LIN {X 0,Y 425.288,Z 130.32,A -85,B 0,C 180,E1 -9761.958,E2 -9761.958} C_VEL
LIN {X 0,Y 425.283,Z 130.319,A -85,B 0,C 180,E1 -9765.283,E2 -9765.283} C_VEL
LIN {X 0,Y 425.272,Z 130.322,A -85,B 0,C 180,E1 -9768.622,E2 -9768.622} C_VEL
LIN {X 0,Y 425.304,Z 130.316,A -85,B 0,C 180,E1 -9771.102,E2 -9771.102} C_VEL
LIN {X 0,Y 425.298,Z 130.317,A -85,B 0,C 180,E1 -9774.664,E2 -9774.664} C_VEL
LIN {X 0,Y 425.263,Z 130.324,A -85,B 0,C 180,E1 -9778.073,E2 -9778.073} C_VEL
LIN {X 0,Y 425.33,Z 130.317,A -85,B 0,C 180,E1 -9781.368,E2 -9781.368} C_VEL
LIN {X 0,Y 425.295,Z 130.314,A -85,B 0,C 180,E1 -9784.555,E2 -9784.555} C_VEL
LIN {X 0,Y 425.395,Z 130.501,A -85,B 0,C 180,E1 -9786.124,E2 -9786.124} C_VEL
LIN {X 0,Y 426.718,Z 138.86,A -85,B 0,C 180,E1 -9788.249,E2 -9788.249} C_VEL
LIN {X 0,Y 426.399,Z 147.655,A -85,B 0,C 180,E1 -9790.343,E2 -9790.343} C_VEL
LIN {X 0,Y 425.564,Z 164.044,A -85,B 0,C 180,E1 -9794.188,E2 -9794.188} C_VEL
LIN {X 0,Y 425.386,Z 168.668,A -85,B 0,C 180,E1 -9795.224,E2 -9795.224} C_VEL
LIN {X 0,Y 425.881,Z 172.494,A -85,B 0,C 180,E1 -9795.359,E2 -9795.359} C_VEL
LIN {X 0,Y 428.081,Z 189.094,A -85,B 0,C 180,E1 -9795.717,E2 -9795.717} C_VEL
LIN {X 0,Y 427.768,Z 244.774,A -85,B 0,C 180,E1 -9796.671,E2 -9796.671} C_VEL
LIN {X 0,Y 427.448,Z 254.051,A -85,B 0,C 180,E1 -9796.934,E2 -9796.934} C_VEL
LIN {X 0,Y 427.1,Z 263.713,A -85,B 0,C 180,E1 -9797.346,E2 -9797.346} C_VEL
LIN {X 0,Y 426.691,Z 272.874,A -85,B 0,C 180,E1 -9797.878,E2 -9797.878} C_VEL
LIN {X 0,Y 426.182,Z 283.679,A -85,B 0,C 180,E1 -9798.707,E2 -9798.707} C_VEL
LIN {X 0,Y 425.644,Z 292.988,A -85,B 0,C 180,E1 -9799.656,E2 -9799.656} C_VEL
LIN {X 0,Y 425.305,Z 299.661,A -85,B 0,C 180,E1 -9800.489,E2 -9800.489} C_VEL
LIN {X 0,Y 424.937,Z 305.994,A -85,B 0,C 180,E1 -9801.44,E2 -9801.44} C_VEL
LIN {X 0,Y 424.669,Z 311.256,A -85,B 0,C 180,E1 -9802.392,E2 -9802.392} C_VEL
LIN {X 0,Y 424.421,Z 316.205,A -85,B 0,C 180,E1 -9803.484,E2 -9803.484} C_VEL
LIN {X 0,Y 424.283,Z 320.82,A -85,B 0,C 180,E1 -9804.773,E2 -9804.773} C_VEL
LIN {X 0,Y 424.129,Z 324.618,A -85,B 0,C 180,E1 -9806.2,E2 -9806.2} C_VEL
LIN {X 0,Y 424.106,Z 326.365,A -85,B 0,C 180,E1 -9807.151,E2 -9807.151} C_VEL
LIN {X 0,Y 424.122,Z 327.617,A -85,B 0,C 180,E1 -9808.101,E2 -9808.101} C_VEL
LIN {X 0,Y 424.067,Z 328.395,A -85,B 0,C 180,E1 -9809.051,E2 -9809.051} C_VEL
LIN {X 0,Y 424.06,Z 328.689,A -85,B 0,C 180,E1 -9810,E2 -9810} C_VEL
LIN {X 0,Y 424.067,Z 328.392,A -85,B 0,C 180,E1 -9810.95,E2 -9810.95} C_VEL
LIN {X 0,Y 424.122,Z 327.61,A -85,B 0,C 180,E1 -9811.899,E2 -9811.899} C_VEL
LIN {X 0,Y 424.106,Z 326.354,A -85,B 0,C 180,E1 -9812.85,E2 -9812.85} C_VEL
LIN {X 0,Y 424.165,Z 323.448,A -85,B 0,C 180,E1 -9814.276,E2 -9814.276} C_VEL
LIN {X 0,Y 424.283,Z 320.8,A -85,B 0,C 180,E1 -9815.227,E2 -9815.227} C_VEL
LIN {X 0,Y 424.459,Z 315.617,A -85,B 0,C 180,E1 -9816.656,E2 -9816.656} C_VEL
LIN {X 0,Y 424.748,Z 308.788,A -85,B 0,C 180,E1 -9818.085,E2 -9818.085} C_VEL
LIN {X 0,Y 425.194,Z 301.324,A -85,B 0,C 180,E1 -9819.274,E2 -9819.274} C_VEL
LIN {X 0,Y 425.588,Z 293.962,A -85,B 0,C 180,E1 -9820.226,E2 -9820.226} C_VEL
LIN {X 0,Y 426.052,Z 286.079,A -85,B 0,C 180,E1 -9821.056,E2 -9821.056} C_VEL
LIN {X 0,Y 426.49,Z 277.748,A -85,B 0,C 180,E1 -9821.767,E2 -9821.767} C_VEL
LIN {X 0,Y 426.99,Z 267.109,A -85,B 0,C 180,E1 -9822.476,E2 -9822.476} C_VEL
LIN {X 0,Y 427.37,Z 255.53,A -85,B 0,C 180,E1 -9823.008,E2 -9823.008} C_VEL
LIN {X 0,Y 427.68,Z 245.835,A -85,B 0,C 180,E1 -9823.301,E2 -9823.301} C_VEL
LIN {X 0,Y 428.097,Z 188.695,A -85,B 0,C 180,E1 -9824.283,E2 -9824.283} C_VEL
LIN {X 0,Y 425.376,Z 168.966,A -85,B 0,C 180,E1 -9824.74,E2 -9824.74} C_VEL
LIN {X 0,Y 425.469,Z 166.107,A -85,B 0,C 180,E1 -9825.325,E2 -9825.325} C_VEL
LIN {X 0,Y 426.143,Z 151.434,A -85,B 0,C 180,E1 -9828.76,E2 -9828.76} C_VEL
LIN {X 0,Y 426.783,Z 139.882,A -85,B 0,C 180,E1 -9831.494,E2 -9831.494} C_VEL
LIN {X 0,Y 426.048,Z 134.247,A -85,B 0,C 180,E1 -9832.894,E2 -9832.894} C_VEL
LIN {X 0,Y 425.366,Z 130.353,A -85,B 0,C 180,E1 -9833.943,E2 -9833.943} C_VEL
LIN {X 0,Y 425.349,Z 130.31,A -85,B 0,C 180,E1 -9837.558,E2 -9837.558} C_VEL
LIN {X 0,Y 425.288,Z 130.32,A -85,B 0,C 180,E1 -9840.816,E2 -9840.816} C_VEL
LIN {X 0,Y 425.312,Z 130.321,A -85,B 0,C 180,E1 -9844.288,E2 -9844.288} C_VEL
LIN {X 0,Y 425.279,Z 130.322,A -85,B 0,C 180,E1 -9847.694,E2 -9847.694} C_VEL
LIN {X 0,Y 425.28,Z 130.32,A -85,B 0,C 180,E1 -9850.52,E2 -9850.52} C_VEL
LIN {X 0,Y 425.257,Z 130.324,A -85,B 0,C 180,E1 -9853.351,E2 -9853.351} C_VEL
LIN {X 0,Y 425.257,Z 130.322,A -85,B 0,C 180,E1 -9856.649,E2 -9856.649} C_VEL
LIN {X 0,Y 425.286,Z 130.322,A -85,B 0,C 180,E1 -9859.873,E2 -9859.873} C_VEL
LIN {X 0,Y 425.278,Z 130.319,A -85,B 0,C 180,E1 -9862.489,E2 -9862.489} C_VEL
LIN {X 0,Y 425.309,Z 130.317,A -85,B 0,C 180,E1 -9865.818,E2 -9865.818} C_VEL
LIN {X 0,Y 425.291,Z 130.325,A -85,B 0,C 180,E1 -9869.239,E2 -9869.239} C_VEL
LIN {X 0,Y 425.35,Z 130.311,A -85,B 0,C 180,E1 -9872.442,E2 -9872.442} C_VEL
LIN {X 0,Y 425.352,Z 130.311,A -85,B 0,C 180,E1 -9875.602,E2 -9875.602} C_VEL
LIN {X 0,Y 425.294,Z 130.322,A -85,B 0,C 180,E1 -9878.682,E2 -9878.682} C_VEL
LIN {X 0,Y 425.334,Z 130.312,A -85,B 0,C 180,E1 -9881.703,E2 -9881.703} C_VEL
LIN {X 0,Y 425.35,Z 130.317,A -85,B 0,C 180,E1 -9884.671,E2 -9884.671} C_VEL
LIN {X 0,Y 425.413,Z 130.302,A -85,B 0,C 180,E1 -9887.598,E2 -9887.598} C_VEL
LIN {X 0,Y 425.444,Z 130.298,A -85,B 0,C 180,E1 -9891.45,E2 -9891.45} C_VEL
LIN {X 0,Y 425.552,Z 130.292,A -85,B 0,C 180,E1 -9894.313,E2 -9894.313} C_VEL
LIN {X 0,Y 425.575,Z 130.289,A -85,B 0,C 180,E1 -9898.107,E2 -9898.107} C_VEL
LIN {X 0,Y 425.703,Z 130.273,A -85,B 0,C 180,E1 -9900,E2 -9900} C_VEL
LIN {X 0,Y 425.547,Z 130.286,A -85,B 0,C 180,E1 -9902.84,E2 -9902.84} C_VEL
LIN {X 0,Y 425.533,Z 130.288,A -85,B 0,C 180,E1 -9906.639,E2 -9906.639} C_VEL
LIN {X 0,Y 425.405,Z 130.308,A -85,B 0,C 180,E1 -9909.509,E2 -9909.509} C_VEL
LIN {X 0,Y 425.406,Z 130.304,A -85,B 0,C 180,E1 -9912.91,E2 -9912.91} C_VEL
LIN {X 0,Y 425.363,Z 130.309,A -85,B 0,C 180,E1 -9916.605,E2 -9916.605} C_VEL
LIN {X 0,Y 425.33,Z 130.316,A -85,B 0,C 180,E1 -9919.636,E2 -9919.636} C_VEL
LIN {X 0,Y 425.308,Z 130.32,A -85,B 0,C 180,E1 -9923.365,E2 -9923.365} C_VEL
LIN {X 0,Y 425.349,Z 130.315,A -85,B 0,C 180,E1 -9926.844,E2 -9926.844} C_VEL
LIN {X 0,Y 425.293,Z 130.318,A -85,B 0,C 180,E1 -9929.72,E2 -9929.72} C_VEL
LIN {X 0,Y 425.284,Z 130.323,A -85,B 0,C 180,E1 -9933.048,E2 -9933.048} C_VEL
LIN {X 0,Y 425.285,Z 130.319,A -85,B 0,C 180,E1 -9935.929,E2 -9935.929} C_VEL
LIN {X 0,Y 425.283,Z 130.321,A -85,B 0,C 180,E1 -9939.041,E2 -9939.041} C_VEL
LIN {X 0,Y 425.291,Z 130.319,A -85,B 0,C 180,E1 -9941.958,E2 -9941.958} C_VEL
LIN {X 0,Y 425.286,Z 130.318,A -85,B 0,C 180,E1 -9945.283,E2 -9945.283} C_VEL
LIN {X 0,Y 425.277,Z 130.322,A -85,B 0,C 180,E1 -9948.622,E2 -9948.622} C_VEL
LIN {X 0,Y 425.317,Z 130.314,A -85,B 0,C 180,E1 -9951.103,E2 -9951.103} C_VEL
LIN {X 0,Y 425.302,Z 130.317,A -85,B 0,C 180,E1 -9954.664,E2 -9954.664} C_VEL
LIN {X 0,Y 425.267,Z 130.325,A -85,B 0,C 180,E1 -9958.073,E2 -9958.073} C_VEL
LIN {X 0,Y 425.333,Z 130.315,A -85,B 0,C 180,E1 -9961.368,E2 -9961.368} C_VEL
LIN {X 0,Y 425.355,Z 130.315,A -85,B 0,C 180,E1 -9963.505,E2 -9963.505} C_VEL
LIN {X 0,Y 425.287,Z 130.321,A -85,B 0,C 180,E1 -9966.634,E2 -9966.634} C_VEL
LIN {X 0,Y 425.375,Z 130.436,A -85,B 0,C 180,E1 -9969.13,E2 -9969.13} C_VEL
LIN {X 0,Y 426.152,Z 136.277,A -85,B 0,C 180,E1 -9970.741,E2 -9970.741} C_VEL
LIN {X 0,Y 425.734,Z 147.759,A -85,B 0,C 180,E1 -9973.702,E2 -9973.702} C_VEL
LIN {X 0,Y 425.508,Z 154.307,A -85,B 0,C 180,E1 -9975.298,E2 -9975.298} C_VEL
LIN {X 0,Y 426.018,Z 157.356,A -85,B 0,C 180,E1 -9975.412,E2 -9975.412} C_VEL
LIN {X 0,Y 428.175,Z 170.829,A -85,B 0,C 180,E1 -9975.717,E2 -9975.717} C_VEL
LIN {X 0,Y 427.787,Z 230.137,A -85,B 0,C 180,E1 -9976.733,E2 -9976.733} C_VEL
LIN {X 0,Y 427.576,Z 239.219,A -85,B 0,C 180,E1 -9976.998,E2 -9976.998} C_VEL
LIN {X 0,Y 427.327,Z 248.804,A -85,B 0,C 180,E1 -9977.413,E2 -9977.413} C_VEL
LIN {X 0,Y 426.923,Z 258.842,A -85,B 0,C 180,E1 -9978.004,E2 -9978.004} C_VEL
LIN {X 0,Y 426.381,Z 269.256,A -85,B 0,C 180,E1 -9978.833,E2 -9978.833} C_VEL
LIN {X 0,Y 425.985,Z 277.399,A -85,B 0,C 180,E1 -9979.664,E2 -9979.664} C_VEL
LIN {X 0,Y 425.58,Z 284.118,A -85,B 0,C 180,E1 -9980.494,E2 -9980.494} C_VEL
LIN {X 0,Y 425.466,Z 285.604,A -85,B 0,C 180,E1 -9980.702,E2 -9980.702} C_VEL
LIN {X 0,Y 424.548,Z 289.624,A -85,B 0,C 180,E1 -9981.28,E2 -9981.28} C_VEL
LIN {X 0,Y 420.037,Z 297.702,A -85,B 0,C 180,E1 -9982.687,E2 -9982.687} C_VEL
LIN {X 0,Y 417.925,Z 301.654,A -85,B 0,C 180,E1 -9983.579,E2 -9983.579} C_VEL
LIN {X 0,Y 417.506,Z 303.441,A -85,B 0,C 180,E1 -9984.055,E2 -9984.055} C_VEL
LIN {X 0,Y 417.267,Z 306.984,A -85,B 0,C 180,E1 -9985.169,E2 -9985.169} C_VEL
LIN {X 0,Y 417.172,Z 309.308,A -85,B 0,C 180,E1 -9986.136,E2 -9986.136} C_VEL
LIN {X 0,Y 417.127,Z 311.078,A -85,B 0,C 180,E1 -9987.102,E2 -9987.102} C_VEL
LIN {X 0,Y 417.064,Z 312.355,A -85,B 0,C 180,E1 -9988.068,E2 -9988.068} C_VEL
LIN {X 0,Y 416.993,Z 313.163,A -85,B 0,C 180,E1 -9989.034,E2 -9989.034} C_VEL
LIN {X 0,Y 416.983,Z 313.47,A -85,B 0,C 180,E1 -9990,E2 -9990} C_VEL
LIN {X 0,Y 416.993,Z 313.195,A -85,B 0,C 180,E1 -9990.965,E2 -9990.965} C_VEL
LIN {X 0,Y 417.064,Z 312.452,A -85,B 0,C 180,E1 -9991.931,E2 -9991.931} C_VEL
LIN {X 0,Y 417.125,Z 311.241,A -85,B 0,C 180,E1 -9992.897,E2 -9992.897} C_VEL
LIN {X 0,Y 417.2,Z 308.392,A -85,B 0,C 180,E1 -9994.347,E2 -9994.347} C_VEL
LIN {X 0,Y 417.362,Z 305.799,A -85,B 0,C 180,E1 -9995.314,E2 -9995.314} C_VEL
LIN {X 0,Y 417.669,Z 300.692,A -85,B 0,C 180,E1 -9996.764,E2 -9996.764} C_VEL
LIN {X 0,Y 417.888,Z 295.199,A -85,B 0,C 180,E1 -9997.975,E2 -9997.975} C_VEL
LIN {X 0,Y 418.33,Z 288.3,A -85,B 0,C 180,E1 -9999.183,E2 -9999.183} C_VEL
LIN {X 0,Y 418.819,Z 280.376,A -85,B 0,C 180,E1 -10000.27,E2 -10000.27} C_VEL
LIN {X 0,Y 419.251,Z 272.82,A -85,B 0,C 180,E1 -10001.115,E2 -10001.115} C_VEL
LIN {X 0,Y 419.666,Z 264.901,A -85,B 0,C 180,E1 -10001.838,E2 -10001.838} C_VEL
LIN {X 0,Y 420.075,Z 256.724,A -85,B 0,C 180,E1 -10002.439,E2 -10002.439} C_VEL
LIN {X 0,Y 420.443,Z 248.443,A -85,B 0,C 180,E1 -10002.919,E2 -10002.919} C_VEL
LIN {X 0,Y 420.771,Z 239.505,A -85,B 0,C 180,E1 -10003.308,E2 -10003.308} C_VEL
LIN {X 0,Y 420.957,Z 230.241,A -85,B 0,C 180,E1 -10003.585,E2 -10003.585} C_VEL
LIN {X 0,Y 421.276,Z 170.679,A -85,B 0,C 180,E1 -10004.626,E2 -10004.626} C_VEL
LIN {X 0,Y 418.531,Z 154.749,A -85,B 0,C 180,E1 -10005.024,E2 -10005.024} C_VEL
LIN {X 0,Y 418.508,Z 153.569,A -85,B 0,C 180,E1 -10005.211,E2 -10005.211} C_VEL
LIN {X 0,Y 419.078,Z 140.565,A -85,B 0,C 180,E1 -10008.58,E2 -10008.58} C_VEL
LIN {X 0,Y 418.969,Z 135.057,A -85,B 0,C 180,E1 -10010.053,E2 -10010.053} C_VEL
LIN {X 0,Y 418.322,Z 131.28,A -85,B 0,C 180,E1 -10011.174,E2 -10011.174} C_VEL
LIN {X 0,Y 418.285,Z 131.193,A -85,B 0,C 180,E1 -10014.864,E2 -10014.864} C_VEL
LIN {X 0,Y 418.292,Z 131.193,A -85,B 0,C 180,E1 -10018.063,E2 -10018.063} C_VEL
LIN {X 0,Y 418.211,Z 131.2,A -85,B 0,C 180,E1 -10021.396,E2 -10021.396} C_VEL
LIN {X 0,Y 418.266,Z 131.195,A -85,B 0,C 180,E1 -10024.58,E2 -10024.58} C_VEL
LIN {X 0,Y 418.234,Z 131.202,A -85,B 0,C 180,E1 -10027.834,E2 -10027.834} C_VEL
LIN {X 0,Y 418.223,Z 131.198,A -85,B 0,C 180,E1 -10030.948,E2 -10030.948} C_VEL
LIN {X 0,Y 418.21,Z 131.207,A -85,B 0,C 180,E1 -10033.729,E2 -10033.729} C_VEL
LIN {X 0,Y 418.207,Z 131.2,A -85,B 0,C 180,E1 -10036.448,E2 -10036.448} C_VEL
LIN {X 0,Y 418.222,Z 131.201,A -85,B 0,C 180,E1 -10039.13,E2 -10039.13} C_VEL
LIN {X 0,Y 418.225,Z 131.198,A -85,B 0,C 180,E1 -10042.167,E2 -10042.167} C_VEL
LIN {X 0,Y 418.265,Z 131.198,A -85,B 0,C 180,E1 -10045.419,E2 -10045.419} C_VEL
LIN {X 0,Y 418.21,Z 131.201,A -85,B 0,C 180,E1 -10048.604,E2 -10048.604} C_VEL
LIN {X 0,Y 418.29,Z 131.19,A -85,B 0,C 180,E1 -10051.936,E2 -10051.936} C_VEL
LIN {X 0,Y 418.288,Z 131.194,A -85,B 0,C 180,E1 -10055.162,E2 -10055.162} C_VEL
LIN {X 0,Y 418.233,Z 131.199,A -85,B 0,C 180,E1 -10058.303,E2 -10058.303} C_VEL
LIN {X 0,Y 418.282,Z 131.191,A -85,B 0,C 180,E1 -10061.383,E2 -10061.383} C_VEL
LIN {X 0,Y 418.301,Z 131.193,A -85,B 0,C 180,E1 -10064.406,E2 -10064.406} C_VEL
LIN {X 0,Y 418.369,Z 131.18,A -85,B 0,C 180,E1 -10067.386,E2 -10067.386} C_VEL
LIN {X 0,Y 418.358,Z 131.188,A -85,B 0,C 180,E1 -10070.329,E2 -10070.329} C_VEL
LIN {X 0,Y 418.493,Z 131.164,A -85,B 0,C 180,E1 -10073.249,E2 -10073.249} C_VEL
LIN {X 0,Y 418.338,Z 131.184,A -85,B 0,C 180,E1 -10075.181,E2 -10075.181} C_VEL
LIN {X 0,Y 418.543,Z 131.165,A -85,B 0,C 180,E1 -10078.075,E2 -10078.075} C_VEL
LIN {X 0,Y 418.671,Z 131.149,A -85,B 0,C 180,E1 -10080,E2 -10080} C_VEL
LIN {X 0,Y 418.5,Z 131.163,A -85,B 0,C 180,E1 -10082.888,E2 -10082.888} C_VEL
LIN {X 0,Y 418.528,Z 131.167,A -85,B 0,C 180,E1 -10085.782,E2 -10085.782} C_VEL
LIN {X 0,Y 418.398,Z 131.176,A -85,B 0,C 180,E1 -10088.695,E2 -10088.695} C_VEL
LIN {X 0,Y 418.314,Z 131.193,A -85,B 0,C 180,E1 -10091.631,E2 -10091.631} C_VEL
LIN {X 0,Y 418.301,Z 131.188,A -85,B 0,C 180,E1 -10094.597,E2 -10094.597} C_VEL
LIN {X 0,Y 418.286,Z 131.194,A -85,B 0,C 180,E1 -10097.604,E2 -10097.604} C_VEL
LIN {X 0,Y 418.248,Z 131.197,A -85,B 0,C 180,E1 -10100.663,E2 -10100.663} C_VEL
LIN {X 0,Y 418.286,Z 131.191,A -85,B 0,C 180,E1 -10103.781,E2 -10103.781} C_VEL
LIN {X 0,Y 418.308,Z 131.193,A -85,B 0,C 180,E1 -10107.071,E2 -10107.071} C_VEL
LIN {X 0,Y 418.242,Z 131.197,A -85,B 0,C 180,E1 -10110.272,E2 -10110.272} C_VEL
LIN {X 0,Y 418.247,Z 131.195,A -85,B 0,C 180,E1 -10113.677,E2 -10113.677} C_VEL
LIN {X 0,Y 418.238,Z 131.197,A -85,B 0,C 180,E1 -10117.224,E2 -10117.224} C_VEL
LIN {X 0,Y 418.242,Z 131.196,A -85,B 0,C 180,E1 -10119.683,E2 -10119.683} C_VEL
LIN {X 0,Y 418.228,Z 131.204,A -85,B 0,C 180,E1 -10122.321,E2 -10122.321} C_VEL
LIN {X 0,Y 418.234,Z 131.197,A -85,B 0,C 180,E1 -10125.109,E2 -10125.109} C_VEL
LIN {X 0,Y 418.238,Z 131.199,A -85,B 0,C 180,E1 -10127.767,E2 -10127.767} C_VEL
LIN {X 0,Y 418.251,Z 131.196,A -85,B 0,C 180,E1 -10130.62,E2 -10130.62} C_VEL
LIN {X 0,Y 418.242,Z 131.202,A -85,B 0,C 180,E1 -10133.976,E2 -10133.976} C_VEL
LIN {X 0,Y 418.256,Z 131.195,A -85,B 0,C 180,E1 -10137.156,E2 -10137.156} C_VEL
LIN {X 0,Y 418.267,Z 131.193,A -85,B 0,C 180,E1 -10140.896,E2 -10140.896} C_VEL
LIN {X 0,Y 418.27,Z 131.195,A -85,B 0,C 180,E1 -10144.096,E2 -10144.096} C_VEL
LIN {X 0,Y 418.338,Z 131.267,A -85,B 0,C 180,E1 -10145.893,E2 -10145.893} C_VEL
LIN {X 0,Y 419.711,Z 139.787,A -85,B 0,C 180,E1 -10148.126,E2 -10148.126} C_VEL
LIN {X 0,Y 419.509,Z 146.454,A -85,B 0,C 180,E1 -10149.745,E2 -10149.745} C_VEL
LIN {X 0,Y 418.631,Z 161.823,A -85,B 0,C 180,E1 -10153.418,E2 -10153.418} C_VEL
LIN {X 0,Y 418.359,Z 168.541,A -85,B 0,C 180,E1 -10154.97,E2 -10154.97} C_VEL
LIN {X 0,Y 418.92,Z 172.639,A -85,B 0,C 180,E1 -10155.114,E2 -10155.114} C_VEL
LIN {X 0,Y 421.205,Z 189.538,A -85,B 0,C 180,E1 -10155.488,E2 -10155.488} C_VEL
LIN {X 0,Y 420.872,Z 244.708,A -85,B 0,C 180,E1 -10156.45,E2 -10156.45} C_VEL
LIN {X 0,Y 420.552,Z 253.932,A -85,B 0,C 180,E1 -10156.716,E2 -10156.716} C_VEL
LIN {X 0,Y 420.184,Z 263.592,A -85,B 0,C 180,E1 -10157.135,E2 -10157.135} C_VEL
LIN {X 0,Y 419.759,Z 272.751,A -85,B 0,C 180,E1 -10157.674,E2 -10157.674} C_VEL
LIN {X 0,Y 419.186,Z 283.554,A -85,B 0,C 180,E1 -10158.516,E2 -10158.516} C_VEL
LIN {X 0,Y 418.668,Z 292.863,A -85,B 0,C 180,E1 -10159.482,E2 -10159.482} C_VEL
LIN {X 0,Y 418.275,Z 299.534,A -85,B 0,C 180,E1 -10160.327,E2 -10160.327} C_VEL
LIN {X 0,Y 417.889,Z 305.867,A -85,B 0,C 180,E1 -10161.294,E2 -10161.294} C_VEL
LIN {X 0,Y 417.609,Z 311.129,A -85,B 0,C 180,E1 -10162.263,E2 -10162.263} C_VEL
LIN {X 0,Y 417.344,Z 316.535,A -85,B 0,C 180,E1 -10163.488,E2 -10163.488} C_VEL
LIN {X 0,Y 417.202,Z 320.692,A -85,B 0,C 180,E1 -10164.684,E2 -10164.684} C_VEL
LIN {X 0,Y 417.092,Z 323.336,A -85,B 0,C 180,E1 -10165.652,E2 -10165.652} C_VEL
LIN {X 0,Y 417.005,Z 326.237,A -85,B 0,C 180,E1 -10167.102,E2 -10167.102} C_VEL
LIN {X 0,Y 417.031,Z 327.489,A -85,B 0,C 180,E1 -10168.069,E2 -10168.069} C_VEL
LIN {X 0,Y 416.99,Z 328.267,A -85,B 0,C 180,E1 -10169.035,E2 -10169.035} C_VEL
LIN {X 0,Y 416.981,Z 328.561,A -85,B 0,C 180,E1 -10170,E2 -10170} C_VEL
LIN {X 0,Y 416.99,Z 328.264,A -85,B 0,C 180,E1 -10170.966,E2 -10170.966} C_VEL
LIN {X 0,Y 417.031,Z 327.482,A -85,B 0,C 180,E1 -10171.932,E2 -10171.932} C_VEL
LIN {X 0,Y 417.005,Z 326.225,A -85,B 0,C 180,E1 -10172.898,E2 -10172.898} C_VEL
LIN {X 0,Y 417.092,Z 323.319,A -85,B 0,C 180,E1 -10174.349,E2 -10174.349} C_VEL
LIN {X 0,Y 417.202,Z 320.67,A -85,B 0,C 180,E1 -10175.316,E2 -10175.316} C_VEL
LIN {X 0,Y 417.344,Z 316.507,A -85,B 0,C 180,E1 -10176.512,E2 -10176.512} C_VEL
LIN {X 0,Y 417.546,Z 311.089,A -85,B 0,C 180,E1 -10177.739,E2 -10177.739} C_VEL
LIN {X 0,Y 417.97,Z 304.402,A -85,B 0,C 180,E1 -10178.948,E2 -10178.948} C_VEL
LIN {X 0,Y 418.468,Z 295.876,A -85,B 0,C 180,E1 -10180.157,E2 -10180.157} C_VEL
LIN {X 0,Y 419.03,Z 287.179,A -85,B 0,C 180,E1 -10181.121,E2 -10181.121} C_VEL
LIN {X 0,Y 419.459,Z 279.118,A -85,B 0,C 180,E1 -10181.844,E2 -10181.844} C_VEL
LIN {X 0,Y 419.871,Z 270.764,A -85,B 0,C 180,E1 -10182.446,E2 -10182.446} C_VEL
LIN {X 0,Y 420.228,Z 262.236,A -85,B 0,C 180,E1 -10182.926,E2 -10182.926} C_VEL
LIN {X 0,Y 420.549,Z 252.897,A -85,B 0,C 180,E1 -10183.315,E2 -10183.315} C_VEL
LIN {X 0,Y 420.88,Z 241.831,A -85,B 0,C 180,E1 -10183.611,E2 -10183.611} C_VEL
LIN {X 0,Y 421.104,Z 187.899,A -85,B 0,C 180,E1 -10184.537,E2 -10184.537} C_VEL
LIN {X 0,Y 418.388,Z 169.009,A -85,B 0,C 180,E1 -10184.979,E2 -10184.979} C_VEL
LIN {X 0,Y 418.402,Z 167.128,A -85,B 0,C 180,E1 -10185.316,E2 -10185.316} C_VEL
LIN {X 0,Y 419.137,Z 152.355,A -85,B 0,C 180,E1 -10188.831,E2 -10188.831} C_VEL
LIN {X 0,Y 419.79,Z 140.808,A -85,B 0,C 180,E1 -10191.612,E2 -10191.612} C_VEL
LIN {X 0,Y 418.524,Z 132.329,A -85,B 0,C 180,E1 -10193.767,E2 -10193.767} C_VEL
LIN {X 0,Y 418.321,Z 131.178,A -85,B 0,C 180,E1 -10194.174,E2 -10194.174} C_VEL
LIN {X 0,Y 418.311,Z 131.188,A -85,B 0,C 180,E1 -10197.071,E2 -10197.071} C_VEL
LIN {X 0,Y 418.245,Z 131.202,A -85,B 0,C 180,E1 -10200.272,E2 -10200.272} C_VEL
LIN {X 0,Y 418.249,Z 131.196,A -85,B 0,C 180,E1 -10203.677,E2 -10203.677} C_VEL
LIN {X 0,Y 418.24,Z 131.196,A -85,B 0,C 180,E1 -10207.224,E2 -10207.224} C_VEL
LIN {X 0,Y 418.249,Z 131.199,A -85,B 0,C 180,E1 -10209.682,E2 -10209.682} C_VEL
LIN {X 0,Y 418.23,Z 131.199,A -85,B 0,C 180,E1 -10212.321,E2 -10212.321} C_VEL
LIN {X 0,Y 418.236,Z 131.197,A -85,B 0,C 180,E1 -10215.109,E2 -10215.109} C_VEL
LIN {X 0,Y 418.24,Z 131.202,A -85,B 0,C 180,E1 -10217.767,E2 -10217.767} C_VEL
LIN {X 0,Y 418.246,Z 131.195,A -85,B 0,C 180,E1 -10220.621,E2 -10220.621} C_VEL
LIN {X 0,Y 418.245,Z 131.197,A -85,B 0,C 180,E1 -10223.976,E2 -10223.976} C_VEL
LIN {X 0,Y 418.258,Z 131.199,A -85,B 0,C 180,E1 -10227.156,E2 -10227.156} C_VEL
LIN {X 0,Y 418.269,Z 131.196,A -85,B 0,C 180,E1 -10230.896,E2 -10230.896} C_VEL
LIN {X 0,Y 418.272,Z 131.192,A -85,B 0,C 180,E1 -10234.096,E2 -10234.096} C_VEL
LIN {X 0,Y 418.239,Z 131.199,A -85,B 0,C 180,E1 -10237.264,E2 -10237.264} C_VEL
LIN {X 0,Y 418.285,Z 131.193,A -85,B 0,C 180,E1 -10240.364,E2 -10240.364} C_VEL
LIN {X 0,Y 418.319,Z 131.187,A -85,B 0,C 180,E1 -10243.405,E2 -10243.405} C_VEL
LIN {X 0,Y 418.348,Z 131.185,A -85,B 0,C 180,E1 -10246.999,E2 -10246.999} C_VEL
LIN {X 0,Y 418.342,Z 131.189,A -85,B 0,C 180,E1 -10250.329,E2 -10250.329} C_VEL
LIN {X 0,Y 418.49,Z 131.165,A -85,B 0,C 180,E1 -10253.249,E2 -10253.249} C_VEL
LIN {X 0,Y 418.339,Z 131.184,A -85,B 0,C 180,E1 -10255.182,E2 -10255.182} C_VEL
LIN {X 0,Y 418.544,Z 131.164,A -85,B 0,C 180,E1 -10258.076,E2 -10258.076} C_VEL
LIN {X 0,Y 418.672,Z 131.148,A -85,B 0,C 180,E1 -10260,E2 -10260} C_VEL
LIN {X 0,Y 418.502,Z 131.163,A -85,B 0,C 180,E1 -10262.888,E2 -10262.888} C_VEL
LIN {X 0,Y 418.495,Z 131.164,A -85,B 0,C 180,E1 -10266.751,E2 -10266.751} C_VEL
LIN {X 0,Y 418.361,Z 131.188,A -85,B 0,C 180,E1 -10269.671,E2 -10269.671} C_VEL
LIN {X 0,Y 418.357,Z 131.183,A -85,B 0,C 180,E1 -10273.006,E2 -10273.006} C_VEL
LIN {X 0,Y 418.315,Z 131.187,A -85,B 0,C 180,E1 -10276.736,E2 -10276.736} C_VEL
LIN {X 0,Y 418.272,Z 131.194,A -85,B 0,C 180,E1 -10279.79,E2 -10279.79} C_VEL
LIN {X 0,Y 418.24,Z 131.198,A -85,B 0,C 180,E1 -10282.736,E2 -10282.736} C_VEL
LIN {X 0,Y 418.272,Z 131.192,A -85,B 0,C 180,E1 -10285.904,E2 -10285.904} C_VEL
LIN {X 0,Y 418.266,Z 131.197,A -85,B 0,C 180,E1 -10289.162,E2 -10289.162} C_VEL
LIN {X 0,Y 418.259,Z 131.201,A -85,B 0,C 180,E1 -10292.844,E2 -10292.844} C_VEL
LIN {X 0,Y 418.247,Z 131.197,A -85,B 0,C 180,E1 -10296.238,E2 -10296.238} C_VEL
LIN {X 0,Y 418.246,Z 131.195,A -85,B 0,C 180,E1 -10299.683,E2 -10299.683} C_VEL
LIN {X 0,Y 418.231,Z 131.202,A -85,B 0,C 180,E1 -10302.321,E2 -10302.321} C_VEL
LIN {X 0,Y 418.237,Z 131.197,A -85,B 0,C 180,E1 -10305.109,E2 -10305.109} C_VEL
LIN {X 0,Y 418.242,Z 131.197,A -85,B 0,C 180,E1 -10307.767,E2 -10307.767} C_VEL
LIN {X 0,Y 418.262,Z 131.195,A -85,B 0,C 180,E1 -10310.618,E2 -10310.618} C_VEL
LIN {X 0,Y 418.248,Z 131.201,A -85,B 0,C 180,E1 -10313.976,E2 -10313.976} C_VEL
LIN {X 0,Y 418.259,Z 131.194,A -85,B 0,C 180,E1 -10317.156,E2 -10317.156} C_VEL
LIN {X 0,Y 418.27,Z 131.192,A -85,B 0,C 180,E1 -10320.895,E2 -10320.895} C_VEL
LIN {X 0,Y 418.27,Z 131.194,A -85,B 0,C 180,E1 -10324.096,E2 -10324.096} C_VEL
LIN {X 0,Y 418.234,Z 131.201,A -85,B 0,C 180,E1 -10327.263,E2 -10327.263} C_VEL
LIN {X 0,Y 418.349,Z 131.416,A -85,B 0,C 180,E1 -10329.02,E2 -10329.02} C_VEL
LIN {X 0,Y 419.121,Z 136.368,A -85,B 0,C 180,E1 -10330.405,E2 -10330.405} C_VEL
LIN {X 0,Y 418.816,Z 146.391,A -85,B 0,C 180,E1 -10333.038,E2 -10333.038} C_VEL
LIN {X 0,Y 418.527,Z 154.432,A -85,B 0,C 180,E1 -10335.047,E2 -10335.047} C_VEL
LIN {X 0,Y 419.069,Z 157.734,A -85,B 0,C 180,E1 -10335.168,E2 -10335.168} C_VEL
LIN {X 0,Y 421.319,Z 171.168,A -85,B 0,C 180,E1 -10335.482,E2 -10335.482} C_VEL
LIN {X 0,Y 420.876,Z 230.284,A -85,B 0,C 180,E1 -10336.511,E2 -10336.511} C_VEL
LIN {X 0,Y 420.682,Z 239.36,A -85,B 0,C 180,E1 -10336.781,E2 -10336.781} C_VEL
LIN {X 0,Y 420.428,Z 248.941,A -85,B 0,C 180,E1 -10337.203,E2 -10337.203} C_VEL
LIN {X 0,Y 420.023,Z 257.108,A -85,B 0,C 180,E1 -10337.682,E2 -10337.682} C_VEL
LIN {X 0,Y 419.558,Z 266.705,A -85,B 0,C 180,E1 -10338.404,E2 -10338.404} C_VEL
LIN {X 0,Y 419.075,Z 276.512,A -85,B 0,C 180,E1 -10339.369,E2 -10339.369} C_VEL
LIN {X 0,Y 418.592,Z 284.249,A -85,B 0,C 180,E1 -10340.334,E2 -10340.334} C_VEL
LIN {X 0,Y 418.147,Z 290.61,A -85,B 0,C 180,E1 -10341.299,E2 -10341.299} C_VEL
LIN {X 0,Y 417.809,Z 297.066,A -85,B 0,C 180,E1 -10342.509,E2 -10342.509} C_VEL
LIN {X 0,Y 417.594,Z 302.214,A -85,B 0,C 180,E1 -10343.719,E2 -10343.719} C_VEL
LIN {X 0,Y 417.506,Z 303.441,A -85,B 0,C 180,E1 -10344.055,E2 -10344.055} C_VEL
LIN {X 0,Y 416.696,Z 305.939,A -85,B 0,C 180,E1 -10344.782,E2 -10344.782} C_VEL
LIN {X 0,Y 413.688,Z 309.302,A -85,B 0,C 180,E1 -10346.002,E2 -10346.002} C_VEL
LIN {X 0,Y 411.19,Z 311.256,A -85,B 0,C 180,E1 -10347.018,E2 -10347.018} C_VEL
LIN {X 0,Y 410.082,Z 312.281,A -85,B 0,C 180,E1 -10347.82,E2 -10347.82} C_VEL
LIN {X 0,Y 409.971,Z 312.532,A -85,B 0,C 180,E1 -10348.093,E2 -10348.093} C_VEL
LIN {X 0,Y 409.919,Z 313.291,A -85,B 0,C 180,E1 -10349.017,E2 -10349.017} C_VEL
LIN {X 0,Y 409.906,Z 313.598,A -85,B 0,C 180,E1 -10350,E2 -10350} C_VEL
LIN {X 0,Y 409.919,Z 313.323,A -85,B 0,C 180,E1 -10350.982,E2 -10350.982} C_VEL
LIN {X 0,Y 409.978,Z 312.58,A -85,B 0,C 180,E1 -10351.965,E2 -10351.965} C_VEL
LIN {X 0,Y 410.028,Z 311.368,A -85,B 0,C 180,E1 -10352.947,E2 -10352.947} C_VEL
LIN {X 0,Y 410.124,Z 308.519,A -85,B 0,C 180,E1 -10354.422,E2 -10354.422} C_VEL
LIN {X 0,Y 410.308,Z 305.926,A -85,B 0,C 180,E1 -10355.405,E2 -10355.405} C_VEL
LIN {X 0,Y 410.526,Z 302.179,A -85,B 0,C 180,E1 -10356.53,E2 -10356.53} C_VEL
LIN {X 0,Y 410.734,Z 297.781,A -85,B 0,C 180,E1 -10357.595,E2 -10357.595} C_VEL
LIN {X 0,Y 410.999,Z 292.719,A -85,B 0,C 180,E1 -10358.605,E2 -10358.605} C_VEL
LIN {X 0,Y 411.428,Z 286.749,A -85,B 0,C 180,E1 -10359.587,E2 -10359.587} C_VEL
LIN {X 0,Y 411.895,Z 279.482,A -85,B 0,C 180,E1 -10360.569,E2 -10360.569} C_VEL
LIN {X 0,Y 412.384,Z 271.716,A -85,B 0,C 180,E1 -10361.427,E2 -10361.427} C_VEL
LIN {X 0,Y 412.862,Z 263.524,A -85,B 0,C 180,E1 -10362.16,E2 -10362.16} C_VEL
LIN {X 0,Y 413.218,Z 254.975,A -85,B 0,C 180,E1 -10362.774,E2 -10362.774} C_VEL
LIN {X 0,Y 413.775,Z 243.662,A -85,B 0,C 180,E1 -10363.381,E2 -10363.381} C_VEL
LIN {X 0,Y 414.021,Z 233.216,A -85,B 0,C 180,E1 -10363.748,E2 -10363.748} C_VEL
LIN {X 0,Y 414.152,Z 214.748,A -85,B 0,C 180,E1 -10364.111,E2 -10364.111} C_VEL
LIN {X 0,Y 414.447,Z 171.804,A -85,B 0,C 180,E1 -10364.854,E2 -10364.854} C_VEL
LIN {X 0,Y 411.558,Z 154.862,A -85,B 0,C 180,E1 -10365.284,E2 -10365.284} C_VEL
LIN {X 0,Y 411.495,Z 153.69,A -85,B 0,C 180,E1 -10365.477,E2 -10365.477} C_VEL
LIN {X 0,Y 412.023,Z 142.585,A -85,B 0,C 180,E1 -10368.394,E2 -10368.394} C_VEL
LIN {X 0,Y 412.042,Z 136.841,A -85,B 0,C 180,E1 -10369.945,E2 -10369.945} C_VEL
LIN {X 0,Y 411.285,Z 132.183,A -85,B 0,C 180,E1 -10371.291,E2 -10371.291} C_VEL
LIN {X 0,Y 411.236,Z 132.069,A -85,B 0,C 180,E1 -10375.293,E2 -10375.293} C_VEL
LIN {X 0,Y 411.259,Z 132.066,A -85,B 0,C 180,E1 -10377.477,E2 -10377.477} C_VEL
LIN {X 0,Y 411.189,Z 132.075,A -85,B 0,C 180,E1 -10380.847,E2 -10380.847} C_VEL
LIN {X 0,Y 411.206,Z 132.076,A -85,B 0,C 180,E1 -10384.333,E2 -10384.333} C_VEL
LIN {X 0,Y 411.2,Z 132.08,A -85,B 0,C 180,E1 -10387.973,E2 -10387.973} C_VEL
LIN {X 0,Y 411.183,Z 132.076,A -85,B 0,C 180,E1 -10390.504,E2 -10390.504} C_VEL
LIN {X 0,Y 411.173,Z 132.077,A -85,B 0,C 180,E1 -10393.133,E2 -10393.133} C_VEL
LIN {X 0,Y 411.167,Z 132.081,A -85,B 0,C 180,E1 -10395.881,E2 -10395.881} C_VEL
LIN {X 0,Y 411.162,Z 132.078,A -85,B 0,C 180,E1 -10398.771,E2 -10398.771} C_VEL
LIN {X 0,Y 411.191,Z 132.075,A -85,B 0,C 180,E1 -10402.026,E2 -10402.026} C_VEL
LIN {X 0,Y 411.205,Z 132.075,A -85,B 0,C 180,E1 -10405.666,E2 -10405.666} C_VEL
LIN {X 0,Y 411.188,Z 132.081,A -85,B 0,C 180,E1 -10409.152,E2 -10409.152} C_VEL
LIN {X 0,Y 411.258,Z 132.067,A -85,B 0,C 180,E1 -10412.522,E2 -10412.522} C_VEL
LIN {X 0,Y 411.225,Z 132.07,A -85,B 0,C 180,E1 -10415.784,E2 -10415.784} C_VEL
LIN {X 0,Y 411.195,Z 132.078,A -85,B 0,C 180,E1 -10418.966,E2 -10418.966} C_VEL
LIN {X 0,Y 411.251,Z 132.068,A -85,B 0,C 180,E1 -10422.085,E2 -10422.085} C_VEL
LIN {X 0,Y 411.261,Z 132.066,A -85,B 0,C 180,E1 -10425.147,E2 -10425.147} C_VEL
LIN {X 0,Y 411.298,Z 132.065,A -85,B 0,C 180,E1 -10428.168,E2 -10428.168} C_VEL
LIN {X 0,Y 411.48,Z 132.043,A -85,B 0,C 180,E1 -10432.147,E2 -10432.147} C_VEL
LIN {X 0,Y 411.474,Z 132.045,A -85,B 0,C 180,E1 -10434.118,E2 -10434.118} C_VEL
LIN {X 0,Y 411.512,Z 132.041,A -85,B 0,C 180,E1 -10438.042,E2 -10438.042} C_VEL
LIN {X 0,Y 411.641,Z 132.025,A -85,B 0,C 180,E1 -10440,E2 -10440} C_VEL
LIN {X 0,Y 411.457,Z 132.041,A -85,B 0,C 180,E1 -10442.937,E2 -10442.937} C_VEL
LIN {X 0,Y 411.487,Z 132.043,A -85,B 0,C 180,E1 -10445.882,E2 -10445.882} C_VEL
LIN {X 0,Y 411.48,Z 132.043,A -85,B 0,C 180,E1 -10447.853,E2 -10447.853} C_VEL
LIN {X 0,Y 411.282,Z 132.066,A -85,B 0,C 180,E1 -10451.833,E2 -10451.833} C_VEL
LIN {X 0,Y 411.258,Z 132.067,A -85,B 0,C 180,E1 -10454.853,E2 -10454.853} C_VEL
LIN {X 0,Y 411.251,Z 132.068,A -85,B 0,C 180,E1 -10457.915,E2 -10457.915} C_VEL
LIN {X 0,Y 411.195,Z 132.079,A -85,B 0,C 180,E1 -10461.034,E2 -10461.034} C_VEL
LIN {X 0,Y 411.225,Z 132.07,A -85,B 0,C 180,E1 -10464.215,E2 -10464.215} C_VEL
LIN {X 0,Y 411.257,Z 132.067,A -85,B 0,C 180,E1 -10467.478,E2 -10467.478} C_VEL
LIN {X 0,Y 411.188,Z 132.081,A -85,B 0,C 180,E1 -10470.848,E2 -10470.848} C_VEL
LIN {X 0,Y 411.204,Z 132.076,A -85,B 0,C 180,E1 -10474.334,E2 -10474.334} C_VEL
LIN {X 0,Y 411.19,Z 132.076,A -85,B 0,C 180,E1 -10477.974,E2 -10477.974} C_VEL
LIN {X 0,Y 411.161,Z 132.078,A -85,B 0,C 180,E1 -10481.228,E2 -10481.228} C_VEL
LIN {X 0,Y 411.174,Z 132.081,A -85,B 0,C 180,E1 -10484.491,E2 -10484.491} C_VEL
LIN {X 0,Y 411.175,Z 132.082,A -85,B 0,C 180,E1 -10488.195,E2 -10488.195} C_VEL
LIN {X 0,Y 411.215,Z 132.071,A -85,B 0,C 180,E1 -10490.776,E2 -10490.776} C_VEL
LIN {X 0,Y 411.197,Z 132.074,A -85,B 0,C 180,E1 -10494.472,E2 -10494.472} C_VEL
LIN {X 0,Y 411.206,Z 132.072,A -85,B 0,C 180,E1 -10496.874,E2 -10496.874} C_VEL
LIN {X 0,Y 411.232,Z 132.069,A -85,B 0,C 180,E1 -10500.644,E2 -10500.644} C_VEL
LIN {X 0,Y 411.237,Z 132.076,A -85,B 0,C 180,E1 -10503.619,E2 -10503.619} C_VEL
LIN {X 0,Y 411.289,Z 132.176,A -85,B 0,C 180,E1 -10505.727,E2 -10505.727} C_VEL
LIN {X 0,Y 412.698,Z 140.714,A -85,B 0,C 180,E1 -10507.998,E2 -10507.998} C_VEL
LIN {X 0,Y 412.516,Z 147.568,A -85,B 0,C 180,E1 -10509.694,E2 -10509.694} C_VEL
LIN {X 0,Y 411.614,Z 162.743,A -85,B 0,C 180,E1 -10513.382,E2 -10513.382} C_VEL
LIN {X 0,Y 411.372,Z 168.414,A -85,B 0,C 180,E1 -10514.709,E2 -10514.709} C_VEL
LIN {X 0,Y 411.875,Z 172.129,A -85,B 0,C 180,E1 -10514.847,E2 -10514.847} C_VEL
LIN {X 0,Y 414.367,Z 190.484,A -85,B 0,C 180,E1 -10515.262,E2 -10515.262} C_VEL
LIN {X 0,Y 413.978,Z 244.646,A -85,B 0,C 180,E1 -10516.221,E2 -10516.221} C_VEL
LIN {X 0,Y 413.666,Z 253.813,A -85,B 0,C 180,E1 -10516.491,E2 -10516.491} C_VEL
LIN {X 0,Y 413.268,Z 263.47,A -85,B 0,C 180,E1 -10516.916,E2 -10516.916} C_VEL
LIN {X 0,Y 412.808,Z 272.627,A -85,B 0,C 180,E1 -10517.463,E2 -10517.463} C_VEL
LIN {X 0,Y 412.206,Z 283.428,A -85,B 0,C 180,E1 -10518.319,E2 -10518.319} C_VEL
LIN {X 0,Y 411.757,Z 291.715,A -85,B 0,C 180,E1 -10519.179,E2 -10519.179} C_VEL
LIN {X 0,Y 411.256,Z 299.407,A -85,B 0,C 180,E1 -10520.161,E2 -10520.161} C_VEL
LIN {X 0,Y 410.843,Z 305.739,A -85,B 0,C 180,E1 -10521.144,E2 -10521.144} C_VEL
LIN {X 0,Y 410.571,Z 311.002,A -85,B 0,C 180,E1 -10522.129,E2 -10522.129} C_VEL
LIN {X 0,Y 410.34,Z 315.39,A -85,B 0,C 180,E1 -10523.114,E2 -10523.114} C_VEL
LIN {X 0,Y 410.14,Z 319.042,A -85,B 0,C 180,E1 -10524.099,E2 -10524.099} C_VEL
LIN {X 0,Y 410.082,Z 322.039,A -85,B 0,C 180,E1 -10525.085,E2 -10525.085} C_VEL
LIN {X 0,Y 409.962,Z 324.363,A -85,B 0,C 180,E1 -10526.068,E2 -10526.068} C_VEL
LIN {X 0,Y 409.905,Z 326.109,A -85,B 0,C 180,E1 -10527.052,E2 -10527.052} C_VEL
LIN {X 0,Y 409.943,Z 327.361,A -85,B 0,C 180,E1 -10528.035,E2 -10528.035} C_VEL
LIN {X 0,Y 409.916,Z 328.139,A -85,B 0,C 180,E1 -10529.018,E2 -10529.018} C_VEL
LIN {X 0,Y 409.904,Z 328.433,A -85,B 0,C 180,E1 -10530,E2 -10530} C_VEL
LIN {X 0,Y 409.916,Z 328.136,A -85,B 0,C 180,E1 -10530.983,E2 -10530.983} C_VEL
LIN {X 0,Y 409.943,Z 327.353,A -85,B 0,C 180,E1 -10531.965,E2 -10531.965} C_VEL
LIN {X 0,Y 409.905,Z 326.096,A -85,B 0,C 180,E1 -10532.949,E2 -10532.949} C_VEL
LIN {X 0,Y 410.022,Z 323.19,A -85,B 0,C 180,E1 -10534.424,E2 -10534.424} C_VEL
LIN {X 0,Y 410.124,Z 320.541,A -85,B 0,C 180,E1 -10535.408,E2 -10535.408} C_VEL
LIN {X 0,Y 410.239,Z 316.966,A -85,B 0,C 180,E1 -10536.473,E2 -10536.473} C_VEL
LIN {X 0,Y 410.42,Z 312.134,A -85,B 0,C 180,E1 -10537.626,E2 -10537.626} C_VEL
LIN {X 0,Y 410.742,Z 307.111,A -85,B 0,C 180,E1 -10538.611,E2 -10538.611} C_VEL
LIN {X 0,Y 411.183,Z 301.062,A -85,B 0,C 180,E1 -10539.593,E2 -10539.593} C_VEL
LIN {X 0,Y 411.588,Z 293.699,A -85,B 0,C 180,E1 -10540.577,E2 -10540.577} C_VEL
LIN {X 0,Y 412.114,Z 285.815,A -85,B 0,C 180,E1 -10541.435,E2 -10541.435} C_VEL
LIN {X 0,Y 412.596,Z 277.483,A -85,B 0,C 180,E1 -10542.169,E2 -10542.169} C_VEL
LIN {X 0,Y 413.12,Z 266.841,A -85,B 0,C 180,E1 -10542.902,E2 -10542.902} C_VEL
LIN {X 0,Y 413.566,Z 255.255,A -85,B 0,C 180,E1 -10543.45,E2 -10543.45} C_VEL
LIN {X 0,Y 413.909,Z 245.551,A -85,B 0,C 180,E1 -10543.752,E2 -10543.752} C_VEL
LIN {X 0,Y 414.271,Z 188.839,A -85,B 0,C 180,E1 -10544.763,E2 -10544.763} C_VEL
LIN {X 0,Y 411.397,Z 168.875,A -85,B 0,C 180,E1 -10545.24,E2 -10545.24} C_VEL
LIN {X 0,Y 411.4,Z 166.997,A -85,B 0,C 180,E1 -10545.583,E2 -10545.583} C_VEL
LIN {X 0,Y 412.283,Z 151.179,A -85,B 0,C 180,E1 -10549.415,E2 -10549.415} C_VEL
LIN {X 0,Y 412.799,Z 141.734,A -85,B 0,C 180,E1 -10551.734,E2 -10551.734} C_VEL
LIN {X 0,Y 411.51,Z 133.257,A -85,B 0,C 180,E1 -10553.93,E2 -10553.93} C_VEL
LIN {X 0,Y 411.268,Z 132.07,A -85,B 0,C 180,E1 -10554.337,E2 -10554.337} C_VEL
LIN {X 0,Y 411.259,Z 132.065,A -85,B 0,C 180,E1 -10557.478,E2 -10557.478} C_VEL
LIN {X 0,Y 411.19,Z 132.076,A -85,B 0,C 180,E1 -10560.848,E2 -10560.848} C_VEL
LIN {X 0,Y 411.207,Z 132.077,A -85,B 0,C 180,E1 -10564.334,E2 -10564.334} C_VEL
LIN {X 0,Y 411.195,Z 132.08,A -85,B 0,C 180,E1 -10567.974,E2 -10567.974} C_VEL
LIN {X 0,Y 411.164,Z 132.078,A -85,B 0,C 180,E1 -10571.228,E2 -10571.228} C_VEL
LIN {X 0,Y 411.176,Z 132.076,A -85,B 0,C 180,E1 -10574.491,E2 -10574.491} C_VEL
LIN {X 0,Y 411.177,Z 132.077,A -85,B 0,C 180,E1 -10578.195,E2 -10578.195} C_VEL
LIN {X 0,Y 411.211,Z 132.072,A -85,B 0,C 180,E1 -10580.775,E2 -10580.775} C_VEL
LIN {X 0,Y 411.199,Z 132.073,A -85,B 0,C 180,E1 -10584.471,E2 -10584.471} C_VEL
LIN {X 0,Y 411.208,Z 132.074,A -85,B 0,C 180,E1 -10586.873,E2 -10586.873} C_VEL
LIN {X 0,Y 411.234,Z 132.07,A -85,B 0,C 180,E1 -10590.644,E2 -10590.644} C_VEL
LIN {X 0,Y 411.239,Z 132.069,A -85,B 0,C 180,E1 -10593.619,E2 -10593.619} C_VEL
LIN {X 0,Y 411.204,Z 132.078,A -85,B 0,C 180,E1 -10596.853,E2 -10596.853} C_VEL
LIN {X 0,Y 411.216,Z 132.071,A -85,B 0,C 180,E1 -10600.051,E2 -10600.051} C_VEL
LIN {X 0,Y 411.264,Z 132.067,A -85,B 0,C 180,E1 -10603.131,E2 -10603.131} C_VEL
LIN {X 0,Y 411.307,Z 132.063,A -85,B 0,C 180,E1 -10606.896,E2 -10606.896} C_VEL
LIN {X 0,Y 411.294,Z 132.065,A -85,B 0,C 180,E1 -10610.161,E2 -10610.161} C_VEL
LIN {X 0,Y 411.454,Z 132.042,A -85,B 0,C 180,E1 -10613.133,E2 -10613.133} C_VEL
LIN {X 0,Y 411.31,Z 132.059,A -85,B 0,C 180,E1 -10615.099,E2 -10615.099} C_VEL
LIN {X 0,Y 411.513,Z 132.04,A -85,B 0,C 180,E1 -10618.043,E2 -10618.043} C_VEL
LIN {X 0,Y 411.642,Z 132.024,A -85,B 0,C 180,E1 -10620,E2 -10620} C_VEL
LIN {X 0,Y 411.459,Z 132.041,A -85,B 0,C 180,E1 -10622.937,E2 -10622.937} C_VEL
LIN {X 0,Y 411.462,Z 132.04,A -85,B 0,C 180,E1 -10626.867,E2 -10626.867} C_VEL
LIN {X 0,Y 411.309,Z 132.065,A -85,B 0,C 180,E1 -10629.838,E2 -10629.838} C_VEL
LIN {X 0,Y 411.315,Z 132.061,A -85,B 0,C 180,E1 -10633.109,E2 -10633.109} C_VEL
LIN {X 0,Y 411.259,Z 132.067,A -85,B 0,C 180,E1 -10636.889,E2 -10636.889} C_VEL
LIN {X 0,Y 411.232,Z 132.07,A -85,B 0,C 180,E1 -10639.987,E2 -10639.987} C_VEL
LIN {X 0,Y 411.205,Z 132.079,A -85,B 0,C 180,E1 -10643.148,E2 -10643.148} C_VEL
LIN {X 0,Y 411.24,Z 132.069,A -85,B 0,C 180,E1 -10646.381,E2 -10646.381} C_VEL
LIN {X 0,Y 411.202,Z 132.073,A -85,B 0,C 180,E1 -10649.713,E2 -10649.713} C_VEL
LIN {X 0,Y 411.208,Z 132.075,A -85,B 0,C 180,E1 -10653.156,E2 -10653.156} C_VEL
LIN {X 0,Y 411.195,Z 132.079,A -85,B 0,C 180,E1 -10656.553,E2 -10656.553} C_VEL
LIN {X 0,Y 411.21,Z 132.072,A -85,B 0,C 180,E1 -10659.727,E2 -10659.727} C_VEL
LIN {X 0,Y 411.174,Z 132.077,A -85,B 0,C 180,E1 -10663.134,E2 -10663.134} C_VEL
LIN {X 0,Y 411.17,Z 132.079,A -85,B 0,C 180,E1 -10665.881,E2 -10665.881} C_VEL
LIN {X 0,Y 411.166,Z 132.079,A -85,B 0,C 180,E1 -10668.771,E2 -10668.771} C_VEL
LIN {X 0,Y 411.213,Z 132.075,A -85,B 0,C 180,E1 -10671.83,E2 -10671.83} C_VEL
LIN {X 0,Y 411.213,Z 132.071,A -85,B 0,C 180,E1 -10675.121,E2 -10675.121} C_VEL
LIN {X 0,Y 411.167,Z 132.083,A -85,B 0,C 180,E1 -10678.003,E2 -10678.003} C_VEL
LIN {X 0,Y 411.22,Z 132.073,A -85,B 0,C 180,E1 -10681.41,E2 -10681.41} C_VEL
LIN {X 0,Y 411.239,Z 132.074,A -85,B 0,C 180,E1 -10683.619,E2 -10683.619} C_VEL
LIN {X 0,Y 411.198,Z 132.076,A -85,B 0,C 180,E1 -10686.852,E2 -10686.852} C_VEL
LIN {X 0,Y 411.296,Z 132.24,A -85,B 0,C 180,E1 -10688.84,E2 -10688.84} C_VEL
LIN {X 0,Y 412.144,Z 138.376,A -85,B 0,C 180,E1 -10690.578,E2 -10690.578} C_VEL
LIN {X 0,Y 411.698,Z 149.918,A -85,B 0,C 180,E1 -10693.64,E2 -10693.64} C_VEL
LIN {X 0,Y 411.531,Z 154.558,A -85,B 0,C 180,E1 -10694.787,E2 -10694.787} C_VEL
LIN {X 0,Y 412.04,Z 157.583,A -85,B 0,C 180,E1 -10694.904,E2 -10694.904} C_VEL
LIN {X 0,Y 414.433,Z 171.965,A -85,B 0,C 180,E1 -10695.247,E2 -10695.247} C_VEL
LIN {X 0,Y 413.984,Z 230.431,A -85,B 0,C 180,E1 -10696.282,E2 -10696.282} C_VEL
LIN {X 0,Y 413.789,Z 239.5,A -85,B 0,C 180,E1 -10696.557,E2 -10696.557} C_VEL
LIN {X 0,Y 413.531,Z 249.078,A -85,B 0,C 180,E1 -10696.986,E2 -10696.986} C_VEL
LIN {X 0,Y 413.085,Z 257.243,A -85,B 0,C 180,E1 -10697.472,E2 -10697.472} C_VEL
LIN {X 0,Y 412.607,Z 266.839,A -85,B 0,C 180,E1 -10698.206,E2 -10698.206} C_VEL
LIN {X 0,Y 412.1,Z 276.644,A -85,B 0,C 180,E1 -10699.187,E2 -10699.187} C_VEL
LIN {X 0,Y 411.58,Z 284.381,A -85,B 0,C 180,E1 -10700.168,E2 -10700.168} C_VEL
LIN {X 0,Y 411.121,Z 290.741,A -85,B 0,C 180,E1 -10701.15,E2 -10701.15} C_VEL
LIN {X 0,Y 410.764,Z 297.196,A -85,B 0,C 180,E1 -10702.38,E2 -10702.38} C_VEL
LIN {X 0,Y 410.505,Z 302.954,A -85,B 0,C 180,E1 -10703.768,E2 -10703.768} C_VEL
LIN {X 0,Y 410.208,Z 307.113,A -85,B 0,C 180,E1 -10705.086,E2 -10705.086} C_VEL
LIN {X 0,Y 410.085,Z 309.437,A -85,B 0,C 180,E1 -10706.069,E2 -10706.069} C_VEL
LIN {X 0,Y 410.031,Z 311.207,A -85,B 0,C 180,E1 -10707.052,E2 -10707.052} C_VEL
LIN {X 0,Y 409.971,Z 312.532,A -85,B 0,C 180,E1 -10708.093,E2 -10708.093} C_VEL
LIN {X 0,Y 409.242,Z 313.268,A -85,B 0,C 180,E1 -10708.91,E2 -10708.91} C_VEL
LIN {X 0,Y 406.359,Z 313.628,A -85,B 0,C 180,E1 -10710.243,E2 -10710.243} C_VEL
LIN {X 0,Y 403.529,Z 313.094,A -85,B 0,C 180,E1 -10711.591,E2 -10711.591} C_VEL
LIN {X 0,Y 402.895,Z 312.196,A -85,B 0,C 180,E1 -10712.421,E2 -10712.421} C_VEL
LIN {X 0,Y 402.993,Z 309.794,A -85,B 0,C 180,E1 -10714,E2 -10714} C_VEL
LIN {X 0,Y 403.236,Z 306.053,A -85,B 0,C 180,E1 -10715.501,E2 -10715.501} C_VEL
LIN {X 0,Y 403.57,Z 300.945,A -85,B 0,C 180,E1 -10717.002,E2 -10717.002} C_VEL
LIN {X 0,Y 403.821,Z 295.452,A -85,B 0,C 180,E1 -10718.255,E2 -10718.255} C_VEL
LIN {X 0,Y 404.32,Z 288.551,A -85,B 0,C 180,E1 -10719.505,E2 -10719.505} C_VEL
LIN {X 0,Y 404.846,Z 280.626,A -85,B 0,C 180,E1 -10720.629,E2 -10720.629} C_VEL
LIN {X 0,Y 405.354,Z 273.067,A -85,B 0,C 180,E1 -10721.501,E2 -10721.501} C_VEL
LIN {X 0,Y 405.82,Z 265.146,A -85,B 0,C 180,E1 -10722.248,E2 -10722.248} C_VEL
LIN {X 0,Y 406.229,Z 256.967,A -85,B 0,C 180,E1 -10722.87,E2 -10722.87} C_VEL
LIN {X 0,Y 406.658,Z 248.682,A -85,B 0,C 180,E1 -10723.365,E2 -10723.365} C_VEL
LIN {X 0,Y 406.984,Z 239.737,A -85,B 0,C 180,E1 -10723.767,E2 -10723.767} C_VEL
LIN {X 0,Y 407.185,Z 230.658,A -85,B 0,C 180,E1 -10724.049,E2 -10724.049} C_VEL
LIN {X 0,Y 407.631,Z 172.743,A -85,B 0,C 180,E1 -10725.094,E2 -10725.094} C_VEL
LIN {X 0,Y 404.548,Z 154.979,A -85,B 0,C 180,E1 -10725.556,E2 -10725.556} C_VEL
LIN {X 0,Y 404.523,Z 153.811,A -85,B 0,C 180,E1 -10725.751,E2 -10725.751} C_VEL
LIN {X 0,Y 405.063,Z 142.689,A -85,B 0,C 180,E1 -10728.722,E2 -10728.722} C_VEL
LIN {X 0,Y 404.902,Z 136.932,A -85,B 0,C 180,E1 -10730.313,E2 -10730.313} C_VEL
LIN {X 0,Y 404.221,Z 133.051,A -85,B 0,C 180,E1 -10731.481,E2 -10731.481} C_VEL
LIN {X 0,Y 404.216,Z 132.943,A -85,B 0,C 180,E1 -10735.296,E2 -10735.296} C_VEL
LIN {X 0,Y 404.196,Z 132.948,A -85,B 0,C 180,E1 -10737.999,E2 -10737.999} C_VEL
LIN {X 0,Y 404.139,Z 132.953,A -85,B 0,C 180,E1 -10741.558,E2 -10741.558} C_VEL
LIN {X 0,Y 404.185,Z 132.947,A -85,B 0,C 180,E1 -10745.016,E2 -10745.016} C_VEL
LIN {X 0,Y 404.159,Z 132.95,A -85,B 0,C 180,E1 -10748.756,E2 -10748.756} C_VEL
LIN {X 0,Y 404.123,Z 132.959,A -85,B 0,C 180,E1 -10751.599,E2 -10751.599} C_VEL
LIN {X 0,Y 404.144,Z 132.952,A -85,B 0,C 180,E1 -10754.522,E2 -10754.522} C_VEL
LIN {X 0,Y 404.135,Z 132.956,A -85,B 0,C 180,E1 -10757.295,E2 -10757.295} C_VEL
LIN {X 0,Y 404.168,Z 132.951,A -85,B 0,C 180,E1 -10759.955,E2 -10759.955} C_VEL
LIN {X 0,Y 404.135,Z 132.957,A -85,B 0,C 180,E1 -10763.125,E2 -10763.125} C_VEL
LIN {X 0,Y 404.144,Z 132.952,A -85,B 0,C 180,E1 -10766.187,E2 -10766.187} C_VEL
LIN {X 0,Y 404.144,Z 132.953,A -85,B 0,C 180,E1 -10769.715,E2 -10769.715} C_VEL
LIN {X 0,Y 404.194,Z 132.951,A -85,B 0,C 180,E1 -10773.123,E2 -10773.123} C_VEL
LIN {X 0,Y 404.176,Z 132.95,A -85,B 0,C 180,E1 -10775.334,E2 -10775.334} C_VEL
LIN {X 0,Y 404.137,Z 132.957,A -85,B 0,C 180,E1 -10778.58,E2 -10778.58} C_VEL
LIN {X 0,Y 404.209,Z 132.944,A -85,B 0,C 180,E1 -10781.762,E2 -10781.762} C_VEL
LIN {X 0,Y 404.207,Z 132.947,A -85,B 0,C 180,E1 -10784.882,E2 -10784.882} C_VEL
LIN {X 0,Y 404.269,Z 132.938,A -85,B 0,C 180,E1 -10787.959,E2 -10787.959} C_VEL
LIN {X 0,Y 404.432,Z 132.921,A -85,B 0,C 180,E1 -10792.099,E2 -10792.099} C_VEL
LIN {X 0,Y 404.423,Z 132.922,A -85,B 0,C 180,E1 -10794.015,E2 -10794.015} C_VEL
LIN {X 0,Y 404.481,Z 132.916,A -85,B 0,C 180,E1 -10798.008,E2 -10798.008} C_VEL
LIN {X 0,Y 404.61,Z 132.901,A -85,B 0,C 180,E1 -10800,E2 -10800} C_VEL
LIN {X 0,Y 404.415,Z 132.918,A -85,B 0,C 180,E1 -10802.988,E2 -10802.988} C_VEL
LIN {X 0,Y 404.433,Z 132.92,A -85,B 0,C 180,E1 -10805.985,E2 -10805.985} C_VEL
LIN {X 0,Y 404.421,Z 132.921,A -85,B 0,C 180,E1 -10807.991,E2 -10807.991} C_VEL
LIN {X 0,Y 404.255,Z 132.94,A -85,B 0,C 180,E1 -10812.041,E2 -10812.041} C_VEL
LIN {X 0,Y 404.205,Z 132.948,A -85,B 0,C 180,E1 -10815.118,E2 -10815.118} C_VEL
LIN {X 0,Y 404.209,Z 132.944,A -85,B 0,C 180,E1 -10818.238,E2 -10818.238} C_VEL
LIN {X 0,Y 404.137,Z 132.957,A -85,B 0,C 180,E1 -10821.419,E2 -10821.419} C_VEL
LIN {X 0,Y 404.175,Z 132.951,A -85,B 0,C 180,E1 -10824.666,E2 -10824.666} C_VEL
LIN {X 0,Y 404.193,Z 132.946,A -85,B 0,C 180,E1 -10828,E2 -10828} C_VEL
LIN {X 0,Y 404.137,Z 132.953,A -85,B 0,C 180,E1 -10831.558,E2 -10831.558} C_VEL
LIN {X 0,Y 404.183,Z 132.95,A -85,B 0,C 180,E1 -10835.016,E2 -10835.016} C_VEL
LIN {X 0,Y 404.148,Z 132.955,A -85,B 0,C 180,E1 -10838.758,E2 -10838.758} C_VEL
LIN {X 0,Y 404.12,Z 132.955,A -85,B 0,C 180,E1 -10841.6,E2 -10841.6} C_VEL
LIN {X 0,Y 404.143,Z 132.956,A -85,B 0,C 180,E1 -10844.522,E2 -10844.522} C_VEL
LIN {X 0,Y 404.135,Z 132.953,A -85,B 0,C 180,E1 -10847.296,E2 -10847.296} C_VEL
LIN {X 0,Y 404.167,Z 132.955,A -85,B 0,C 180,E1 -10849.956,E2 -10849.956} C_VEL
LIN {X 0,Y 404.135,Z 132.953,A -85,B 0,C 180,E1 -10853.125,E2 -10853.125} C_VEL
LIN {X 0,Y 404.144,Z 132.955,A -85,B 0,C 180,E1 -10856.188,E2 -10856.188} C_VEL
LIN {X 0,Y 404.144,Z 132.959,A -85,B 0,C 180,E1 -10859.715,E2 -10859.715} C_VEL
LIN {X 0,Y 404.194,Z 132.948,A -85,B 0,C 180,E1 -10863.123,E2 -10863.123} C_VEL
LIN {X 0,Y 404.242,Z 133.062,A -85,B 0,C 180,E1 -10865.544,E2 -10865.544} C_VEL
LIN {X 0,Y 405.681,Z 141.642,A -85,B 0,C 180,E1 -10867.865,E2 -10867.865} C_VEL
LIN {X 0,Y 405.611,Z 147.45,A -85,B 0,C 180,E1 -10869.334,E2 -10869.334} C_VEL
LIN {X 0,Y 404.633,Z 162.615,A -85,B 0,C 180,E1 -10873.087,E2 -10873.087} C_VEL
LIN {X 0,Y 404.356,Z 168.283,A -85,B 0,C 180,E1 -10874.436,E2 -10874.436} C_VEL
LIN {X 0,Y 404.914,Z 172.226,A -85,B 0,C 180,E1 -10874.583,E2 -10874.583} C_VEL
LIN {X 0,Y 407.516,Z 191.333,A -85,B 0,C 180,E1 -10875.025,E2 -10875.025} C_VEL
LIN {X 0,Y 407.038,Z 245.785,A -85,B 0,C 180,E1 -10876.012,E2 -10876.012} C_VEL
LIN {X 0,Y 406.638,Z 257.019,A -85,B 0,C 180,E1 -10876.38,E2 -10876.38} C_VEL
LIN {X 0,Y 406.087,Z 268.755,A -85,B 0,C 180,E1 -10876.998,E2 -10876.998} C_VEL
LIN {X 0,Y 405.685,Z 277.458,A -85,B 0,C 180,E1 -10877.621,E2 -10877.621} C_VEL
LIN {X 0,Y 405.13,Z 285.767,A -85,B 0,C 180,E1 -10878.366,E2 -10878.366} C_VEL
LIN {X 0,Y 404.625,Z 293.633,A -85,B 0,C 180,E1 -10879.239,E2 -10879.239} C_VEL
LIN {X 0,Y 404.161,Z 300.989,A -85,B 0,C 180,E1 -10880.239,E2 -10880.239} C_VEL
LIN {X 0,Y 403.659,Z 308.45,A -85,B 0,C 180,E1 -10881.49,E2 -10881.49} C_VEL
LIN {X 0,Y 403.28,Z 315.263,A -85,B 0,C 180,E1 -10882.993,E2 -10882.993} C_VEL
LIN {X 0,Y 403.027,Z 320.437,A -85,B 0,C 180,E1 -10884.497,E2 -10884.497} C_VEL
LIN {X 0,Y 402.953,Z 323.081,A -85,B 0,C 180,E1 -10885.499,E2 -10885.499} C_VEL
LIN {X 0,Y 402.807,Z 325.981,A -85,B 0,C 180,E1 -10887,E2 -10887} C_VEL
LIN {X 0,Y 402.84,Z 327.233,A -85,B 0,C 180,E1 -10888.001,E2 -10888.001} C_VEL
LIN {X 0,Y 402.844,Z 328.011,A -85,B 0,C 180,E1 -10889.001,E2 -10889.001} C_VEL
LIN {X 0,Y 402.83,Z 328.305,A -85,B 0,C 180,E1 -10890,E2 -10890} C_VEL
LIN {X 0,Y 402.844,Z 328.008,A -85,B 0,C 180,E1 -10891,E2 -10891} C_VEL
LIN {X 0,Y 402.84,Z 327.224,A -85,B 0,C 180,E1 -10892,E2 -10892} C_VEL
LIN {X 0,Y 402.807,Z 325.966,A -85,B 0,C 180,E1 -10893.001,E2 -10893.001} C_VEL
LIN {X 0,Y 402.953,Z 323.061,A -85,B 0,C 180,E1 -10894.502,E2 -10894.502} C_VEL
LIN {X 0,Y 403.027,Z 320.411,A -85,B 0,C 180,E1 -10895.504,E2 -10895.504} C_VEL
LIN {X 0,Y 403.279,Z 315.227,A -85,B 0,C 180,E1 -10897.007,E2 -10897.007} C_VEL
LIN {X 0,Y 403.622,Z 308.396,A -85,B 0,C 180,E1 -10898.512,E2 -10898.512} C_VEL
LIN {X 0,Y 404.161,Z 300.931,A -85,B 0,C 180,E1 -10899.762,E2 -10899.762} C_VEL
LIN {X 0,Y 404.615,Z 293.568,A -85,B 0,C 180,E1 -10900.762,E2 -10900.762} C_VEL
LIN {X 0,Y 405.159,Z 285.683,A -85,B 0,C 180,E1 -10901.634,E2 -10901.634} C_VEL
LIN {X 0,Y 405.663,Z 277.351,A -85,B 0,C 180,E1 -10902.38,E2 -10902.38} C_VEL
LIN {X 0,Y 406.211,Z 266.707,A -85,B 0,C 180,E1 -10903.125,E2 -10903.125} C_VEL
LIN {X 0,Y 406.683,Z 255.118,A -85,B 0,C 180,E1 -10903.682,E2 -10903.682} C_VEL
LIN {X 0,Y 407.031,Z 245.409,A -85,B 0,C 180,E1 -10903.989,E2 -10903.989} C_VEL
LIN {X 0,Y 407.336,Z 188.954,A -85,B 0,C 180,E1 -10905.015,E2 -10905.015} C_VEL
LIN {X 0,Y 404.427,Z 169.06,A -85,B 0,C 180,E1 -10905.497,E2 -10905.497} C_VEL
LIN {X 0,Y 404.378,Z 167.893,A -85,B 0,C 180,E1 -10905.628,E2 -10905.628} C_VEL
LIN {X 0,Y 405.29,Z 152.099,A -85,B 0,C 180,E1 -10909.5,E2 -10909.5} C_VEL
LIN {X 0,Y 405.797,Z 142.657,A -85,B 0,C 180,E1 -10911.861,E2 -10911.861} C_VEL
LIN {X 0,Y 404.265,Z 133.2,A -85,B 0,C 180,E1 -10914.386,E2 -10914.386} C_VEL
LIN {X 0,Y 404.213,Z 132.915,A -85,B 0,C 180,E1 -10914.663,E2 -10914.663} C_VEL
LIN {X 0,Y 404.196,Z 132.948,A -85,B 0,C 180,E1 -10918,E2 -10918} C_VEL
LIN {X 0,Y 404.14,Z 132.953,A -85,B 0,C 180,E1 -10921.558,E2 -10921.558} C_VEL
LIN {X 0,Y 404.185,Z 132.947,A -85,B 0,C 180,E1 -10925.016,E2 -10925.016} C_VEL
LIN {X 0,Y 404.155,Z 132.951,A -85,B 0,C 180,E1 -10928.757,E2 -10928.757} C_VEL
LIN {X 0,Y 404.123,Z 132.958,A -85,B 0,C 180,E1 -10931.6,E2 -10931.6} C_VEL
LIN {X 0,Y 404.146,Z 132.952,A -85,B 0,C 180,E1 -10934.522,E2 -10934.522} C_VEL
LIN {X 0,Y 404.137,Z 132.955,A -85,B 0,C 180,E1 -10937.296,E2 -10937.296} C_VEL
LIN {X 0,Y 404.169,Z 132.951,A -85,B 0,C 180,E1 -10939.956,E2 -10939.956} C_VEL
LIN {X 0,Y 404.137,Z 132.956,A -85,B 0,C 180,E1 -10943.125,E2 -10943.125} C_VEL
LIN {X 0,Y 404.146,Z 132.952,A -85,B 0,C 180,E1 -10946.188,E2 -10946.188} C_VEL
LIN {X 0,Y 404.147,Z 132.953,A -85,B 0,C 180,E1 -10949.715,E2 -10949.715} C_VEL
LIN {X 0,Y 404.197,Z 132.952,A -85,B 0,C 180,E1 -10953.123,E2 -10953.123} C_VEL
LIN {X 0,Y 404.178,Z 132.951,A -85,B 0,C 180,E1 -10955.335,E2 -10955.335} C_VEL
LIN {X 0,Y 404.14,Z 132.956,A -85,B 0,C 180,E1 -10958.581,E2 -10958.581} C_VEL
LIN {X 0,Y 404.212,Z 132.943,A -85,B 0,C 180,E1 -10961.762,E2 -10961.762} C_VEL
LIN {X 0,Y 404.208,Z 132.948,A -85,B 0,C 180,E1 -10964.882,E2 -10964.882} C_VEL
LIN {X 0,Y 404.258,Z 132.939,A -85,B 0,C 180,E1 -10967.959,E2 -10967.959} C_VEL
LIN {X 0,Y 404.406,Z 132.923,A -85,B 0,C 180,E1 -10972.129,E2 -10972.129} C_VEL
LIN {X 0,Y 404.421,Z 132.921,A -85,B 0,C 180,E1 -10974.015,E2 -10974.015} C_VEL
LIN {X 0,Y 404.482,Z 132.915,A -85,B 0,C 180,E1 -10978.009,E2 -10978.009} C_VEL
LIN {X 0,Y 404.611,Z 132.9,A -85,B 0,C 180,E1 -10980,E2 -10980} C_VEL
LIN {X 0,Y 404.417,Z 132.918,A -85,B 0,C 180,E1 -10982.989,E2 -10982.989} C_VEL
LIN {X 0,Y 404.414,Z 132.918,A -85,B 0,C 180,E1 -10986.987,E2 -10986.987} C_VEL
LIN {X 0,Y 404.272,Z 132.939,A -85,B 0,C 180,E1 -10990.011,E2 -10990.011} C_VEL
LIN {X 0,Y 404.268,Z 132.939,A -85,B 0,C 180,E1 -10993.211,E2 -10993.211} C_VEL
LIN {X 0,Y 404.218,Z 132.945,A -85,B 0,C 180,E1 -10997.007,E2 -10997.007} C_VEL
LIN {X 0,Y 404.165,Z 132.949,A -85,B 0,C 180,E1 -11000.352,E2 -11000.352} C_VEL
LIN {X 0,Y 404.171,Z 132.951,A -85,B 0,C 180,E1 -11003.575,E2 -11003.575} C_VEL
LIN {X 0,Y 404.185,Z 132.947,A -85,B 0,C 180,E1 -11005.766,E2 -11005.766} C_VEL
LIN {X 0,Y 404.197,Z 132.945,A -85,B 0,C 180,E1 -11008,E2 -11008} C_VEL
LIN {X 0,Y 404.141,Z 132.953,A -85,B 0,C 180,E1 -11011.558,E2 -11011.558} C_VEL
LIN {X 0,Y 404.187,Z 132.95,A -85,B 0,C 180,E1 -11015.016,E2 -11015.016} C_VEL
LIN {X 0,Y 404.152,Z 132.956,A -85,B 0,C 180,E1 -11018.757,E2 -11018.757} C_VEL
LIN {X 0,Y 404.124,Z 132.954,A -85,B 0,C 180,E1 -11021.6,E2 -11021.6} C_VEL
LIN {X 0,Y 404.146,Z 132.957,A -85,B 0,C 180,E1 -11024.522,E2 -11024.522} C_VEL
LIN {X 0,Y 404.138,Z 132.953,A -85,B 0,C 180,E1 -11027.296,E2 -11027.296} C_VEL
LIN {X 0,Y 404.171,Z 132.953,A -85,B 0,C 180,E1 -11029.955,E2 -11029.955} C_VEL
LIN {X 0,Y 404.142,Z 132.952,A -85,B 0,C 180,E1 -11033.124,E2 -11033.124} C_VEL
LIN {X 0,Y 404.147,Z 132.956,A -85,B 0,C 180,E1 -11036.188,E2 -11036.188} C_VEL
LIN {X 0,Y 404.147,Z 132.957,A -85,B 0,C 180,E1 -11039.715,E2 -11039.715} C_VEL
LIN {X 0,Y 404.197,Z 132.947,A -85,B 0,C 180,E1 -11043.123,E2 -11043.123} C_VEL
LIN {X 0,Y 404.176,Z 132.952,A -85,B 0,C 180,E1 -11045.334,E2 -11045.334} C_VEL
LIN {X 0,Y 404.224,Z 133.079,A -85,B 0,C 180,E1 -11048.652,E2 -11048.652} C_VEL
LIN {X 0,Y 405.084,Z 138.478,A -85,B 0,C 180,E1 -11050.226,E2 -11050.226} C_VEL
LIN {X 0,Y 404.913,Z 146.362,A -85,B 0,C 180,E1 -11052.369,E2 -11052.369} C_VEL
LIN {X 0,Y 404.527,Z 154.655,A -85,B 0,C 180,E1 -11054.513,E2 -11054.513} C_VEL
LIN {X 0,Y 405.019,Z 157.492,A -85,B 0,C 180,E1 -11054.631,E2 -11054.631} C_VEL
LIN {X 0,Y 407.555,Z 173.071,A -85,B 0,C 180,E1 -11055.009,E2 -11055.009} C_VEL
LIN {X 0,Y 407.108,Z 230.578,A -85,B 0,C 180,E1 -11056.046,E2 -11056.046} C_VEL
LIN {X 0,Y 406.908,Z 239.64,A -85,B 0,C 180,E1 -11056.325,E2 -11056.325} C_VEL
LIN {X 0,Y 406.627,Z 249.215,A -85,B 0,C 180,E1 -11056.761,E2 -11056.761} C_VEL
LIN {X 0,Y 406.14,Z 259.247,A -85,B 0,C 180,E1 -11057.381,E2 -11057.381} C_VEL
LIN {X 0,Y 405.537,Z 269.654,A -85,B 0,C 180,E1 -11058.251,E2 -11058.251} C_VEL
LIN {X 0,Y 405.066,Z 277.795,A -85,B 0,C 180,E1 -11059.124,E2 -11059.124} C_VEL
LIN {X 0,Y 404.591,Z 284.512,A -85,B 0,C 180,E1 -11059.996,E2 -11059.996} C_VEL
LIN {X 0,Y 404.111,Z 290.872,A -85,B 0,C 180,E1 -11060.995,E2 -11060.995} C_VEL
LIN {X 0,Y 403.723,Z 297.326,A -85,B 0,C 180,E1 -11062.246,E2 -11062.246} C_VEL
LIN {X 0,Y 403.464,Z 302.318,A -85,B 0,C 180,E1 -11063.457,E2 -11063.457} C_VEL
LIN {X 0,Y 403.152,Z 307.243,A -85,B 0,C 180,E1 -11064.999,E2 -11064.999} C_VEL
LIN {X 0,Y 403.001,Z 309.567,A -85,B 0,C 180,E1 -11066,E2 -11066} C_VEL
LIN {X 0,Y 402.935,Z 311.336,A -85,B 0,C 180,E1 -11067,E2 -11067} C_VEL
LIN {X 0,Y 402.886,Z 312.674,A -85,B 0,C 180,E1 -11068.077,E2 -11068.077} C_VEL
LIN {X 0,Y 402.847,Z 313.419,A -85,B 0,C 180,E1 -11069,E2 -11069} C_VEL
LIN {X 0,Y 402.832,Z 313.727,A -85,B 0,C 180,E1 -11070,E2 -11070} C_VEL
LIN {X 0,Y 402.847,Z 313.451,A -85,B 0,C 180,E1 -11070.999,E2 -11070.999} C_VEL
LIN {X 0,Y 402.895,Z 312.196,A -85,B 0,C 180,E1 -11072.421,E2 -11072.421} C_VEL
LIN {X 0,Y 402.267,Z 311.14,A -85,B 0,C 180,E1 -11073.245,E2 -11073.245} C_VEL
LIN {X 0,Y 399.523,Z 308.756,A -85,B 0,C 180,E1 -11074.569,E2 -11074.569} C_VEL
LIN {X 0,Y 396.864,Z 305.485,A -85,B 0,C 180,E1 -11075.866,E2 -11075.866} C_VEL
LIN {X 0,Y 396.374,Z 302.916,A -85,B 0,C 180,E1 -11076.634,E2 -11076.634} C_VEL
LIN {X 0,Y 396.658,Z 297.917,A -85,B 0,C 180,E1 -11077.892,E2 -11077.892} C_VEL
LIN {X 0,Y 396.953,Z 292.971,A -85,B 0,C 180,E1 -11078.912,E2 -11078.912} C_VEL
LIN {X 0,Y 397.43,Z 287,A -85,B 0,C 180,E1 -11079.928,E2 -11079.928} C_VEL
LIN {X 0,Y 397.964,Z 279.731,A -85,B 0,C 180,E1 -11080.943,E2 -11080.943} C_VEL
LIN {X 0,Y 398.418,Z 273.191,A -85,B 0,C 180,E1 -11081.704,E2 -11081.704} C_VEL
LIN {X 0,Y 398.908,Z 265.269,A -85,B 0,C 180,E1 -11082.463,E2 -11082.463} C_VEL
LIN {X 0,Y 399.331,Z 257.089,A -85,B 0,C 180,E1 -11083.096,E2 -11083.096} C_VEL
LIN {X 0,Y 399.777,Z 248.801,A -85,B 0,C 180,E1 -11083.599,E2 -11083.599} C_VEL
LIN {X 0,Y 400.097,Z 239.854,A -85,B 0,C 180,E1 -11084.009,E2 -11084.009} C_VEL
LIN {X 0,Y 400.309,Z 230.87,A -85,B 0,C 180,E1 -11084.292,E2 -11084.292} C_VEL
LIN {X 0,Y 400.705,Z 173.085,A -85,B 0,C 180,E1 -11085.356,E2 -11085.356} C_VEL
LIN {X 0,Y 397.56,Z 155.098,A -85,B 0,C 180,E1 -11085.836,E2 -11085.836} C_VEL
LIN {X 0,Y 397.565,Z 153.932,A -85,B 0,C 180,E1 -11086.034,E2 -11086.034} C_VEL
LIN {X 0,Y 398.103,Z 142.792,A -85,B 0,C 180,E1 -11089.062,E2 -11089.062} C_VEL
LIN {X 0,Y 397.822,Z 137.495,A -85,B 0,C 180,E1 -11090.559,E2 -11090.559} C_VEL
LIN {X 0,Y 397.182,Z 133.917,A -85,B 0,C 180,E1 -11091.677,E2 -11091.677} C_VEL
LIN {X 0,Y 397.153,Z 133.823,A -85,B 0,C 180,E1 -11095.512,E2 -11095.512} C_VEL
LIN {X 0,Y 397.123,Z 133.831,A -85,B 0,C 180,E1 -11098.543,E2 -11098.543} C_VEL
LIN {X 0,Y 397.079,Z 133.837,A -85,B 0,C 180,E1 -11102.071,E2 -11102.071} C_VEL
LIN {X 0,Y 397.119,Z 133.828,A -85,B 0,C 180,E1 -11105.503,E2 -11105.503} C_VEL
LIN {X 0,Y 397.133,Z 133.825,A -85,B 0,C 180,E1 -11108.862,E2 -11108.862} C_VEL
LIN {X 0,Y 397.068,Z 133.835,A -85,B 0,C 180,E1 -11112.267,E2 -11112.267} C_VEL
LIN {X 0,Y 397.086,Z 133.832,A -85,B 0,C 180,E1 -11115.068,E2 -11115.068} C_VEL
LIN {X 0,Y 397.065,Z 133.836,A -85,B 0,C 180,E1 -11118.021,E2 -11118.021} C_VEL
LIN {X 0,Y 397.125,Z 133.829,A -85,B 0,C 180,E1 -11121.139,E2 -11121.139} C_VEL
LIN {X 0,Y 397.118,Z 133.827,A -85,B 0,C 180,E1 -11124.496,E2 -11124.496} C_VEL
LIN {X 0,Y 397.077,Z 133.833,A -85,B 0,C 180,E1 -11127.928,E2 -11127.928} C_VEL
LIN {X 0,Y 397.121,Z 133.829,A -85,B 0,C 180,E1 -11131.456,E2 -11131.456} C_VEL
LIN {X 0,Y 397.151,Z 133.825,A -85,B 0,C 180,E1 -11134.487,E2 -11134.487} C_VEL
LIN {X 0,Y 397.108,Z 133.832,A -85,B 0,C 180,E1 -11137.085,E2 -11137.085} C_VEL
LIN {X 0,Y 397.147,Z 133.826,A -85,B 0,C 180,E1 -11140.353,E2 -11140.353} C_VEL
LIN {X 0,Y 397.165,Z 133.821,A -85,B 0,C 180,E1 -11143.553,E2 -11143.553} C_VEL
LIN {X 0,Y 397.227,Z 133.818,A -85,B 0,C 180,E1 -11146.703,E2 -11146.703} C_VEL
LIN {X 0,Y 397.227,Z 133.815,A -85,B 0,C 180,E1 -11149.809,E2 -11149.809} C_VEL
LIN {X 0,Y 397.363,Z 133.798,A -85,B 0,C 180,E1 -11152.888,E2 -11152.888} C_VEL
LIN {X 0,Y 397.253,Z 133.811,A -85,B 0,C 180,E1 -11154.925,E2 -11154.925} C_VEL
LIN {X 0,Y 397.45,Z 133.792,A -85,B 0,C 180,E1 -11157.973,E2 -11157.973} C_VEL
LIN {X 0,Y 397.579,Z 133.776,A -85,B 0,C 180,E1 -11160,E2 -11160} C_VEL
LIN {X 0,Y 397.374,Z 133.795,A -85,B 0,C 180,E1 -11163.041,E2 -11163.041} C_VEL
LIN {X 0,Y 397.383,Z 133.797,A -85,B 0,C 180,E1 -11166.091,E2 -11166.091} C_VEL
LIN {X 0,Y 397.375,Z 133.797,A -85,B 0,C 180,E1 -11168.134,E2 -11168.134} C_VEL
LIN {X 0,Y 397.218,Z 133.815,A -85,B 0,C 180,E1 -11172.258,E2 -11172.258} C_VEL
LIN {X 0,Y 397.178,Z 133.827,A -85,B 0,C 180,E1 -11175.392,E2 -11175.392} C_VEL
LIN {X 0,Y 397.161,Z 133.822,A -85,B 0,C 180,E1 -11178.573,E2 -11178.573} C_VEL
LIN {X 0,Y 397.095,Z 133.831,A -85,B 0,C 180,E1 -11181.818,E2 -11181.818} C_VEL
LIN {X 0,Y 397.155,Z 133.828,A -85,B 0,C 180,E1 -11185.132,E2 -11185.132} C_VEL
LIN {X 0,Y 397.16,Z 133.822,A -85,B 0,C 180,E1 -11187.776,E2 -11187.776} C_VEL
LIN {X 0,Y 397.077,Z 133.838,A -85,B 0,C 180,E1 -11190.882,E2 -11190.882} C_VEL
LIN {X 0,Y 397.124,Z 133.831,A -85,B 0,C 180,E1 -11194.493,E2 -11194.493} C_VEL
LIN {X 0,Y 397.098,Z 133.834,A -85,B 0,C 180,E1 -11198.275,E2 -11198.275} C_VEL
LIN {X 0,Y 397.086,Z 133.833,A -85,B 0,C 180,E1 -11200.909,E2 -11200.909} C_VEL
LIN {X 0,Y 397.099,Z 133.83,A -85,B 0,C 180,E1 -11203.649,E2 -11203.649} C_VEL
LIN {X 0,Y 397.1,Z 133.832,A -85,B 0,C 180,E1 -11206.521,E2 -11206.521} C_VEL
LIN {X 0,Y 397.112,Z 133.831,A -85,B 0,C 180,E1 -11210.423,E2 -11210.423} C_VEL
LIN {X 0,Y 397.107,Z 133.831,A -85,B 0,C 180,E1 -11214.266,E2 -11214.266} C_VEL
LIN {X 0,Y 397.113,Z 133.828,A -85,B 0,C 180,E1 -11216.727,E2 -11216.727} C_VEL
LIN {X 0,Y 397.123,Z 133.827,A -85,B 0,C 180,E1 -11220.296,E2 -11220.296} C_VEL
LIN {X 0,Y 397.193,Z 133.818,A -85,B 0,C 180,E1 -11222.61,E2 -11222.61} C_VEL
LIN {X 0,Y 397.195,Z 133.846,A -85,B 0,C 180,E1 -11225.291,E2 -11225.291} C_VEL
LIN {X 0,Y 398.531,Z 141.514,A -85,B 0,C 180,E1 -11227.446,E2 -11227.446} C_VEL
LIN {X 0,Y 398.833,Z 144.676,A -85,B 0,C 180,E1 -11228.282,E2 -11228.282} C_VEL
LIN {X 0,Y 397.981,Z 157.255,A -85,B 0,C 180,E1 -11231.467,E2 -11231.467} C_VEL
LIN {X 0,Y 397.375,Z 168.157,A -85,B 0,C 180,E1 -11234.156,E2 -11234.156} C_VEL
LIN {X 0,Y 398.001,Z 172.536,A -85,B 0,C 180,E1 -11234.317,E2 -11234.317} C_VEL
LIN {X 0,Y 400.627,Z 191.179,A -85,B 0,C 180,E1 -11234.761,E2 -11234.761} C_VEL
LIN {X 0,Y 400.209,Z 244.516,A -85,B 0,C 180,E1 -11235.739,E2 -11235.739} C_VEL
LIN {X 0,Y 399.895,Z 253.574,A -85,B 0,C 180,E1 -11236.016,E2 -11236.016} C_VEL
LIN {X 0,Y 399.448,Z 263.226,A -85,B 0,C 180,E1 -11236.454,E2 -11236.454} C_VEL
LIN {X 0,Y 398.978,Z 272.381,A -85,B 0,C 180,E1 -11237.021,E2 -11237.021} C_VEL
LIN {X 0,Y 398.331,Z 283.178,A -85,B 0,C 180,E1 -11237.906,E2 -11237.906} C_VEL
LIN {X 0,Y 397.726,Z 292.485,A -85,B 0,C 180,E1 -11238.921,E2 -11238.921} C_VEL
LIN {X 0,Y 397.247,Z 299.155,A -85,B 0,C 180,E1 -11239.81,E2 -11239.81} C_VEL
LIN {X 0,Y 396.809,Z 305.486,A -85,B 0,C 180,E1 -11240.828,E2 -11240.828} C_VEL
LIN {X 0,Y 396.462,Z 310.747,A -85,B 0,C 180,E1 -11241.847,E2 -11241.847} C_VEL
LIN {X 0,Y 396.215,Z 315.135,A -85,B 0,C 180,E1 -11242.868,E2 -11242.868} C_VEL
LIN {X 0,Y 395.996,Z 318.786,A -85,B 0,C 180,E1 -11243.887,E2 -11243.887} C_VEL
LIN {X 0,Y 395.917,Z 321.784,A -85,B 0,C 180,E1 -11244.908,E2 -11244.908} C_VEL
LIN {X 0,Y 395.812,Z 324.108,A -85,B 0,C 180,E1 -11245.927,E2 -11245.927} C_VEL
LIN {X 0,Y 395.714,Z 325.853,A -85,B 0,C 180,E1 -11246.946,E2 -11246.946} C_VEL
LIN {X 0,Y 395.737,Z 327.104,A -85,B 0,C 180,E1 -11247.965,E2 -11247.965} C_VEL
LIN {X 0,Y 395.755,Z 327.883,A -85,B 0,C 180,E1 -11248.983,E2 -11248.983} C_VEL
LIN {X 0,Y 395.758,Z 328.177,A -85,B 0,C 180,E1 -11250,E2 -11250} C_VEL
LIN {X 0,Y 395.755,Z 327.88,A -85,B 0,C 180,E1 -11251.018,E2 -11251.018} C_VEL
LIN {X 0,Y 395.737,Z 327.095,A -85,B 0,C 180,E1 -11252.036,E2 -11252.036} C_VEL
LIN {X 0,Y 395.714,Z 325.837,A -85,B 0,C 180,E1 -11253.054,E2 -11253.054} C_VEL
LIN {X 0,Y 395.885,Z 322.932,A -85,B 0,C 180,E1 -11254.582,E2 -11254.582} C_VEL
LIN {X 0,Y 395.933,Z 320.281,A -85,B 0,C 180,E1 -11255.603,E2 -11255.603} C_VEL
LIN {X 0,Y 396.101,Z 317.017,A -85,B 0,C 180,E1 -11256.622,E2 -11256.622} C_VEL
LIN {X 0,Y 396.311,Z 311.873,A -85,B 0,C 180,E1 -11257.9,E2 -11257.9} C_VEL
LIN {X 0,Y 396.681,Z 306.85,A -85,B 0,C 180,E1 -11258.918,E2 -11258.918} C_VEL
LIN {X 0,Y 397.133,Z 300.8,A -85,B 0,C 180,E1 -11259.936,E2 -11259.936} C_VEL
LIN {X 0,Y 397.65,Z 293.437,A -85,B 0,C 180,E1 -11260.953,E2 -11260.953} C_VEL
LIN {X 0,Y 398.184,Z 285.551,A -85,B 0,C 180,E1 -11261.84,E2 -11261.84} C_VEL
LIN {X 0,Y 398.729,Z 277.218,A -85,B 0,C 180,E1 -11262.599,E2 -11262.599} C_VEL
LIN {X 0,Y 399.314,Z 266.573,A -85,B 0,C 180,E1 -11263.356,E2 -11263.356} C_VEL
LIN {X 0,Y 399.801,Z 254.981,A -85,B 0,C 180,E1 -11263.923,E2 -11263.923} C_VEL
LIN {X 0,Y 400.148,Z 245.266,A -85,B 0,C 180,E1 -11264.235,E2 -11264.235} C_VEL
LIN {X 0,Y 400.62,Z 190.849,A -85,B 0,C 180,E1 -11265.236,E2 -11265.236} C_VEL
LIN {X 0,Y 397.413,Z 168.547,A -85,B 0,C 180,E1 -11265.794,E2 -11265.794} C_VEL
LIN {X 0,Y 397.444,Z 166.631,A -85,B 0,C 180,E1 -11266.171,E2 -11266.171} C_VEL
LIN {X 0,Y 398.417,Z 150.921,A -85,B 0,C 180,E1 -11270.12,E2 -11270.12} C_VEL
LIN {X 0,Y 398.816,Z 143.578,A -85,B 0,C 180,E1 -11271.992,E2 -11271.992} C_VEL
LIN {X 0,Y 397.189,Z 133.942,A -85,B 0,C 180,E1 -11274.641,E2 -11274.641} C_VEL
LIN {X 0,Y 397.163,Z 133.822,A -85,B 0,C 180,E1 -11277.776,E2 -11277.776} C_VEL
LIN {X 0,Y 397.079,Z 133.833,A -85,B 0,C 180,E1 -11280.883,E2 -11280.883} C_VEL
LIN {X 0,Y 397.126,Z 133.829,A -85,B 0,C 180,E1 -11284.493,E2 -11284.493} C_VEL
LIN {X 0,Y 397.103,Z 133.833,A -85,B 0,C 180,E1 -11288.275,E2 -11288.275} C_VEL
LIN {X 0,Y 397.089,Z 133.831,A -85,B 0,C 180,E1 -11290.909,E2 -11290.909} C_VEL
LIN {X 0,Y 397.101,Z 133.834,A -85,B 0,C 180,E1 -11293.649,E2 -11293.649} C_VEL
LIN {X 0,Y 397.102,Z 133.829,A -85,B 0,C 180,E1 -11296.521,E2 -11296.521} C_VEL
LIN {X 0,Y 397.113,Z 133.828,A -85,B 0,C 180,E1 -11300.423,E2 -11300.423} C_VEL
LIN {X 0,Y 397.109,Z 133.828,A -85,B 0,C 180,E1 -11304.266,E2 -11304.266} C_VEL
LIN {X 0,Y 397.115,Z 133.829,A -85,B 0,C 180,E1 -11306.727,E2 -11306.727} C_VEL
LIN {X 0,Y 397.125,Z 133.826,A -85,B 0,C 180,E1 -11310.296,E2 -11310.296} C_VEL
LIN {X 0,Y 397.195,Z 133.819,A -85,B 0,C 180,E1 -11312.61,E2 -11312.61} C_VEL
LIN {X 0,Y 397.134,Z 133.825,A -85,B 0,C 180,E1 -11315.982,E2 -11315.982} C_VEL
LIN {X 0,Y 397.14,Z 133.824,A -85,B 0,C 180,E1 -11319.705,E2 -11319.705} C_VEL
LIN {X 0,Y 397.183,Z 133.824,A -85,B 0,C 180,E1 -11322.845,E2 -11322.845} C_VEL
LIN {X 0,Y 397.23,Z 133.818,A -85,B 0,C 180,E1 -11326.703,E2 -11326.703} C_VEL
LIN {X 0,Y 397.219,Z 133.815,A -85,B 0,C 180,E1 -11329.809,E2 -11329.809} C_VEL
LIN {X 0,Y 397.351,Z 133.799,A -85,B 0,C 180,E1 -11332.888,E2 -11332.888} C_VEL
LIN {X 0,Y 397.254,Z 133.811,A -85,B 0,C 180,E1 -11334.925,E2 -11334.925} C_VEL
LIN {X 0,Y 397.451,Z 133.79,A -85,B 0,C 180,E1 -11337.973,E2 -11337.973} C_VEL
LIN {X 0,Y 397.58,Z 133.776,A -85,B 0,C 180,E1 -11340,E2 -11340} C_VEL
LIN {X 0,Y 397.376,Z 133.795,A -85,B 0,C 180,E1 -11343.042,E2 -11343.042} C_VEL
LIN {X 0,Y 397.366,Z 133.797,A -85,B 0,C 180,E1 -11347.112,E2 -11347.112} C_VEL
LIN {X 0,Y 397.23,Z 133.815,A -85,B 0,C 180,E1 -11350.191,E2 -11350.191} C_VEL
LIN {X 0,Y 397.228,Z 133.817,A -85,B 0,C 180,E1 -11353.321,E2 -11353.321} C_VEL
LIN {X 0,Y 397.184,Z 133.823,A -85,B 0,C 180,E1 -11357.155,E2 -11357.155} C_VEL
LIN {X 0,Y 397.104,Z 133.83,A -85,B 0,C 180,E1 -11360.73,E2 -11360.73} C_VEL
LIN {X 0,Y 397.134,Z 133.825,A -85,B 0,C 180,E1 -11364.018,E2 -11364.018} C_VEL
LIN {X 0,Y 397.196,Z 133.82,A -85,B 0,C 180,E1 -11367.39,E2 -11367.39} C_VEL
LIN {X 0,Y 397.081,Z 133.838,A -85,B 0,C 180,E1 -11370.882,E2 -11370.882} C_VEL
LIN {X 0,Y 397.127,Z 133.83,A -85,B 0,C 180,E1 -11374.493,E2 -11374.493} C_VEL
LIN {X 0,Y 397.101,Z 133.832,A -85,B 0,C 180,E1 -11378.275,E2 -11378.275} C_VEL
LIN {X 0,Y 397.09,Z 133.833,A -85,B 0,C 180,E1 -11380.909,E2 -11380.909} C_VEL
LIN {X 0,Y 397.102,Z 133.829,A -85,B 0,C 180,E1 -11383.649,E2 -11383.649} C_VEL
LIN {X 0,Y 397.104,Z 133.833,A -85,B 0,C 180,E1 -11386.521,E2 -11386.521} C_VEL
LIN {X 0,Y 397.117,Z 133.831,A -85,B 0,C 180,E1 -11390.423,E2 -11390.423} C_VEL
LIN {X 0,Y 397.111,Z 133.832,A -85,B 0,C 180,E1 -11394.265,E2 -11394.265} C_VEL
LIN {X 0,Y 397.116,Z 133.828,A -85,B 0,C 180,E1 -11396.727,E2 -11396.727} C_VEL
LIN {X 0,Y 397.126,Z 133.828,A -85,B 0,C 180,E1 -11400.296,E2 -11400.296} C_VEL
LIN {X 0,Y 397.196,Z 133.817,A -85,B 0,C 180,E1 -11402.61,E2 -11402.61} C_VEL
LIN {X 0,Y 397.13,Z 133.832,A -85,B 0,C 180,E1 -11405.981,E2 -11405.981} C_VEL
LIN {X 0,Y 397.177,Z 133.998,A -85,B 0,C 180,E1 -11408.493,E2 -11408.493} C_VEL
LIN {X 0,Y 398.141,Z 140.498,A -85,B 0,C 180,E1 -11410.404,E2 -11410.404} C_VEL
LIN {X 0,Y 397.775,Z 150.155,A -85,B 0,C 180,E1 -11413.05,E2 -11413.05} C_VEL
LIN {X 0,Y 397.565,Z 154.825,A -85,B 0,C 180,E1 -11414.24,E2 -11414.24} C_VEL
LIN {X 0,Y 398.198,Z 158.661,A -85,B 0,C 180,E1 -11414.38,E2 -11414.38} C_VEL
LIN {X 0,Y 400.762,Z 174.307,A -85,B 0,C 180,E1 -11414.768,E2 -11414.768} C_VEL
LIN {X 0,Y 400.244,Z 230.725,A -85,B 0,C 180,E1 -11415.801,E2 -11415.801} C_VEL
LIN {X 0,Y 399.962,Z 240.612,A -85,B 0,C 180,E1 -11416.115,E2 -11416.115} C_VEL
LIN {X 0,Y 399.607,Z 251.755,A -85,B 0,C 180,E1 -11416.654,E2 -11416.654} C_VEL
LIN {X 0,Y 399.061,Z 262.61,A -85,B 0,C 180,E1 -11417.412,E2 -11417.412} C_VEL
LIN {X 0,Y 398.523,Z 271.015,A -85,B 0,C 180,E1 -11418.17,E2 -11418.17} C_VEL
LIN {X 0,Y 398.028,Z 278.947,A -85,B 0,C 180,E1 -11419.058,E2 -11419.058} C_VEL
LIN {X 0,Y 397.616,Z 284.643,A -85,B 0,C 180,E1 -11419.819,E2 -11419.819} C_VEL
LIN {X 0,Y 397.089,Z 291.003,A -85,B 0,C 180,E1 -11420.834,E2 -11420.834} C_VEL
LIN {X 0,Y 396.673,Z 297.457,A -85,B 0,C 180,E1 -11422.108,E2 -11422.108} C_VEL
LIN {X 0,Y 396.489,Z 301.328,A -85,B 0,C 180,E1 -11423.041,E2 -11423.041} C_VEL
LIN {X 0,Y 396.187,Z 305.885,A -85,B 0,C 180,E1 -11424.401,E2 -11424.401} C_VEL
LIN {X 0,Y 395.994,Z 308.549,A -85,B 0,C 180,E1 -11425.419,E2 -11425.419} C_VEL
LIN {X 0,Y 395.84,Z 311.465,A -85,B 0,C 180,E1 -11426.947,E2 -11426.947} C_VEL
LIN {X 0,Y 395.797,Z 312.741,A -85,B 0,C 180,E1 -11427.965,E2 -11427.965} C_VEL
LIN {X 0,Y 395.76,Z 313.548,A -85,B 0,C 180,E1 -11428.982,E2 -11428.982} C_VEL
LIN {X 0,Y 395.76,Z 313.854,A -85,B 0,C 180,E1 -11430,E2 -11430} C_VEL
LIN {X 0,Y 395.76,Z 313.579,A -85,B 0,C 180,E1 -11431.017,E2 -11431.017} C_VEL
LIN {X 0,Y 395.797,Z 312.366,A -85,B 0,C 180,E1 -11432.429,E2 -11432.429} C_VEL
LIN {X 0,Y 395.915,Z 309.921,A -85,B 0,C 180,E1 -11434.071,E2 -11434.071} C_VEL
LIN {X 0,Y 396.17,Z 306.18,A -85,B 0,C 180,E1 -11435.599,E2 -11435.599} C_VEL
LIN {X 0,Y 396.374,Z 302.916,A -85,B 0,C 180,E1 -11436.634,E2 -11436.634} C_VEL
LIN {X 0,Y 395.897,Z 300.189,A -85,B 0,C 180,E1 -11437.379,E2 -11437.379} C_VEL
LIN {X 0,Y 393.373,Z 295.216,A -85,B 0,C 180,E1 -11438.57,E2 -11438.57} C_VEL
LIN {X 0,Y 390.922,Z 289.539,A -85,B 0,C 180,E1 -11439.704,E2 -11439.704} C_VEL
LIN {X 0,Y 390.572,Z 285.519,A -85,B 0,C 180,E1 -11440.352,E2 -11440.352} C_VEL
LIN {X 0,Y 391.121,Z 277.819,A -85,B 0,C 180,E1 -11441.4,E2 -11441.4} C_VEL
LIN {X 0,Y 391.76,Z 268.351,A -85,B 0,C 180,E1 -11442.431,E2 -11442.431} C_VEL
LIN {X 0,Y 392.344,Z 259.081,A -85,B 0,C 180,E1 -11443.202,E2 -11443.202} C_VEL
LIN {X 0,Y 392.845,Z 250.129,A -85,B 0,C 180,E1 -11443.778,E2 -11443.778} C_VEL
LIN {X 0,Y 393.221,Z 240.801,A -85,B 0,C 180,E1 -11444.226,E2 -11444.226} C_VEL
LIN {X 0,Y 393.444,Z 231.069,A -85,B 0,C 180,E1 -11444.545,E2 -11444.545} C_VEL
LIN {X 0,Y 393.894,Z 174.061,A -85,B 0,C 180,E1 -11445.612,E2 -11445.612} C_VEL
LIN {X 0,Y 390.61,Z 155.112,A -85,B 0,C 180,E1 -11446.134,E2 -11446.134} C_VEL
LIN {X 0,Y 390.551,Z 154.372,A -85,B 0,C 180,E1 -11446.247,E2 -11446.247} C_VEL
LIN {X 0,Y 391.132,Z 142.897,A -85,B 0,C 180,E1 -11449.415,E2 -11449.415} C_VEL
LIN {X 0,Y 390.774,Z 138.321,A -85,B 0,C 180,E1 -11450.737,E2 -11450.737} C_VEL
LIN {X 0,Y 390.142,Z 134.801,A -85,B 0,C 180,E1 -11451.845,E2 -11451.845} C_VEL
LIN {X 0,Y 390.119,Z 134.7,A -85,B 0,C 180,E1 -11455.743,E2 -11455.743} C_VEL
LIN {X 0,Y 390.059,Z 134.707,A -85,B 0,C 180,E1 -11459.109,E2 -11459.109} C_VEL
LIN {X 0,Y 390.043,Z 134.71,A -85,B 0,C 180,E1 -11462.721,E2 -11462.721} C_VEL
LIN {X 0,Y 390.057,Z 134.711,A -85,B 0,C 180,E1 -11465.825,E2 -11465.825} C_VEL
LIN {X 0,Y 390.071,Z 134.706,A -85,B 0,C 180,E1 -11469.218,E2 -11469.218} C_VEL
LIN {X 0,Y 390.042,Z 134.71,A -85,B 0,C 180,E1 -11472.374,E2 -11472.374} C_VEL
LIN {X 0,Y 390.043,Z 134.712,A -85,B 0,C 180,E1 -11475.354,E2 -11475.354} C_VEL
LIN {X 0,Y 390.03,Z 134.711,A -85,B 0,C 180,E1 -11478.186,E2 -11478.186} C_VEL
LIN {X 0,Y 390.086,Z 134.704,A -85,B 0,C 180,E1 -11480.907,E2 -11480.907} C_VEL
LIN {X 0,Y 390.084,Z 134.705,A -85,B 0,C 180,E1 -11484.793,E2 -11484.793} C_VEL
LIN {X 0,Y 390.022,Z 134.712,A -85,B 0,C 180,E1 -11488.495,E2 -11488.495} C_VEL
LIN {X 0,Y 390.116,Z 134.699,A -85,B 0,C 180,E1 -11492.07,E2 -11492.07} C_VEL
LIN {X 0,Y 390.079,Z 134.705,A -85,B 0,C 180,E1 -11495.519,E2 -11495.519} C_VEL
LIN {X 0,Y 390.054,Z 134.713,A -85,B 0,C 180,E1 -11498.878,E2 -11498.878} C_VEL
LIN {X 0,Y 390.127,Z 134.7,A -85,B 0,C 180,E1 -11502.167,E2 -11502.167} C_VEL
LIN {X 0,Y 390.146,Z 134.696,A -85,B 0,C 180,E1 -11505.393,E2 -11505.393} C_VEL
LIN {X 0,Y 390.158,Z 134.699,A -85,B 0,C 180,E1 -11508.571,E2 -11508.571} C_VEL
LIN {X 0,Y 390.343,Z 134.675,A -85,B 0,C 180,E1 -11511.993,E2 -11511.993} C_VEL
LIN {X 0,Y 390.225,Z 134.687,A -85,B 0,C 180,E1 -11514.833,E2 -11514.833} C_VEL
LIN {X 0,Y 390.419,Z 134.667,A -85,B 0,C 180,E1 -11517.937,E2 -11517.937} C_VEL
LIN {X 0,Y 390.549,Z 134.652,A -85,B 0,C 180,E1 -11520,E2 -11520} C_VEL
LIN {X 0,Y 390.309,Z 134.676,A -85,B 0,C 180,E1 -11523.096,E2 -11523.096} C_VEL
LIN {X 0,Y 390.336,Z 134.674,A -85,B 0,C 180,E1 -11526.202,E2 -11526.202} C_VEL
LIN {X 0,Y 390.313,Z 134.676,A -85,B 0,C 180,E1 -11528.282,E2 -11528.282} C_VEL
LIN {X 0,Y 390.169,Z 134.693,A -85,B 0,C 180,E1 -11532.483,E2 -11532.483} C_VEL
LIN {X 0,Y 390.138,Z 134.7,A -85,B 0,C 180,E1 -11535.677,E2 -11535.677} C_VEL
LIN {X 0,Y 390.104,Z 134.704,A -85,B 0,C 180,E1 -11538.922,E2 -11538.922} C_VEL
LIN {X 0,Y 390.038,Z 134.709,A -85,B 0,C 180,E1 -11542.234,E2 -11542.234} C_VEL
LIN {X 0,Y 390.117,Z 134.7,A -85,B 0,C 180,E1 -11545.743,E2 -11545.743} C_VEL
LIN {X 0,Y 390.057,Z 134.711,A -85,B 0,C 180,E1 -11549.11,E2 -11549.11} C_VEL
LIN {X 0,Y 390.041,Z 134.716,A -85,B 0,C 180,E1 -11552.722,E2 -11552.722} C_VEL
LIN {X 0,Y 390.054,Z 134.707,A -85,B 0,C 180,E1 -11555.825,E2 -11555.825} C_VEL
LIN {X 0,Y 390.065,Z 134.706,A -85,B 0,C 180,E1 -11559.218,E2 -11559.218} C_VEL
LIN {X 0,Y 390.041,Z 134.715,A -85,B 0,C 180,E1 -11562.374,E2 -11562.374} C_VEL
LIN {X 0,Y 390.042,Z 134.709,A -85,B 0,C 180,E1 -11565.355,E2 -11565.355} C_VEL
LIN {X 0,Y 390.03,Z 134.716,A -85,B 0,C 180,E1 -11568.187,E2 -11568.187} C_VEL
LIN {X 0,Y 390.088,Z 134.703,A -85,B 0,C 180,E1 -11570.908,E2 -11570.908} C_VEL
LIN {X 0,Y 390.084,Z 134.703,A -85,B 0,C 180,E1 -11574.793,E2 -11574.793} C_VEL
LIN {X 0,Y 390.031,Z 134.715,A -85,B 0,C 180,E1 -11577.876,E2 -11577.876} C_VEL
LIN {X 0,Y 390.057,Z 134.707,A -85,B 0,C 180,E1 -11580.891,E2 -11580.891} C_VEL
LIN {X 0,Y 390.118,Z 134.697,A -85,B 0,C 180,E1 -11584.257,E2 -11584.257} C_VEL
LIN {X 0,Y 390.183,Z 134.87,A -85,B 0,C 180,E1 -11585.172,E2 -11585.172} C_VEL
LIN {X 0,Y 391.796,Z 144.548,A -85,B 0,C 180,E1 -11587.871,E2 -11587.871} C_VEL
LIN {X 0,Y 391.424,Z 151.891,A -85,B 0,C 180,E1 -11589.78,E2 -11589.78} C_VEL
LIN {X 0,Y 390.417,Z 167.684,A -85,B 0,C 180,E1 -11593.799,E2 -11593.799} C_VEL
LIN {X 0,Y 390.418,Z 168.386,A -85,B 0,C 180,E1 -11593.899,E2 -11593.899} C_VEL
LIN {X 0,Y 393.811,Z 192.258,A -85,B 0,C 180,E1 -11594.512,E2 -11594.512} C_VEL
LIN {X 0,Y 393.341,Z 244.453,A -85,B 0,C 180,E1 -11595.486,E2 -11595.486} C_VEL
LIN {X 0,Y 393.02,Z 253.455,A -85,B 0,C 180,E1 -11595.767,E2 -11595.767} C_VEL
LIN {X 0,Y 392.633,Z 261.894,A -85,B 0,C 180,E1 -11596.149,E2 -11596.149} C_VEL
LIN {X 0,Y 392.177,Z 270.383,A -85,B 0,C 180,E1 -11596.66,E2 -11596.66} C_VEL
LIN {X 0,Y 391.741,Z 278.711,A -85,B 0,C 180,E1 -11597.305,E2 -11597.305} C_VEL
LIN {X 0,Y 391.147,Z 286.748,A -85,B 0,C 180,E1 -11598.075,E2 -11598.075} C_VEL
LIN {X 0,Y 390.5,Z 295.426,A -85,B 0,C 180,E1 -11599.107,E2 -11599.107} C_VEL
LIN {X 0,Y 389.917,Z 303.938,A -85,B 0,C 180,E1 -11600.403,E2 -11600.403} C_VEL
LIN {X 0,Y 389.431,Z 310.62,A -85,B 0,C 180,E1 -11601.699,E2 -11601.699} C_VEL
LIN {X 0,Y 389.102,Z 316.062,A -85,B 0,C 180,E1 -11603.023,E2 -11603.023} C_VEL
LIN {X 0,Y 388.844,Z 320.181,A -85,B 0,C 180,E1 -11604.295,E2 -11604.295} C_VEL
LIN {X 0,Y 388.798,Z 322.825,A -85,B 0,C 180,E1 -11605.334,E2 -11605.334} C_VEL
LIN {X 0,Y 388.624,Z 325.725,A -85,B 0,C 180,E1 -11606.89,E2 -11606.89} C_VEL
LIN {X 0,Y 388.635,Z 326.976,A -85,B 0,C 180,E1 -11607.928,E2 -11607.928} C_VEL
LIN {X 0,Y 388.654,Z 327.754,A -85,B 0,C 180,E1 -11608.964,E2 -11608.964} C_VEL
LIN {X 0,Y 388.671,Z 328.049,A -85,B 0,C 180,E1 -11610,E2 -11610} C_VEL
LIN {X 0,Y 388.654,Z 327.751,A -85,B 0,C 180,E1 -11611.036,E2 -11611.036} C_VEL
LIN {X 0,Y 388.635,Z 326.966,A -85,B 0,C 180,E1 -11612.073,E2 -11612.073} C_VEL
LIN {X 0,Y 388.624,Z 325.708,A -85,B 0,C 180,E1 -11613.11,E2 -11613.11} C_VEL
LIN {X 0,Y 388.798,Z 322.802,A -85,B 0,C 180,E1 -11614.666,E2 -11614.666} C_VEL
LIN {X 0,Y 388.844,Z 320.151,A -85,B 0,C 180,E1 -11615.705,E2 -11615.705} C_VEL
LIN {X 0,Y 389.04,Z 316.887,A -85,B 0,C 180,E1 -11616.743,E2 -11616.743} C_VEL
LIN {X 0,Y 389.278,Z 311.743,A -85,B 0,C 180,E1 -11618.043,E2 -11618.043} C_VEL
LIN {X 0,Y 389.666,Z 306.72,A -85,B 0,C 180,E1 -11619.08,E2 -11619.08} C_VEL
LIN {X 0,Y 390.118,Z 300.669,A -85,B 0,C 180,E1 -11620.117,E2 -11620.117} C_VEL
LIN {X 0,Y 390.683,Z 293.305,A -85,B 0,C 180,E1 -11621.15,E2 -11621.15} C_VEL
LIN {X 0,Y 391.217,Z 285.419,A -85,B 0,C 180,E1 -11622.054,E2 -11622.054} C_VEL
LIN {X 0,Y 391.788,Z 277.086,A -85,B 0,C 180,E1 -11622.826,E2 -11622.826} C_VEL
LIN {X 0,Y 392.421,Z 266.439,A -85,B 0,C 180,E1 -11623.595,E2 -11623.595} C_VEL
LIN {X 0,Y 392.92,Z 254.843,A -85,B 0,C 180,E1 -11624.172,E2 -11624.172} C_VEL
LIN {X 0,Y 393.274,Z 245.123,A -85,B 0,C 180,E1 -11624.489,E2 -11624.489} C_VEL
LIN {X 0,Y 393.681,Z 190.483,A -85,B 0,C 180,E1 -11625.515,E2 -11625.515} C_VEL
LIN {X 0,Y 390.408,Z 168.326,A -85,B 0,C 180,E1 -11626.092,E2 -11626.092} C_VEL
LIN {X 0,Y 390.627,Z 163.833,A -85,B 0,C 180,E1 -11627.148,E2 -11627.148} C_VEL
LIN {X 0,Y 391.682,Z 148.484,A -85,B 0,C 180,E1 -11631.086,E2 -11631.086} C_VEL
LIN {X 0,Y 391.65,Z 143.445,A -85,B 0,C 180,E1 -11632.416,E2 -11632.416} C_VEL
LIN {X 0,Y 390.201,Z 135.015,A -85,B 0,C 180,E1 -11634.757,E2 -11634.757} C_VEL
LIN {X 0,Y 390.143,Z 134.674,A -85,B 0,C 180,E1 -11635.045,E2 -11635.045} C_VEL
LIN {X 0,Y 390.097,Z 134.704,A -85,B 0,C 180,E1 -11638.02,E2 -11638.02} C_VEL
LIN {X 0,Y 390.024,Z 134.711,A -85,B 0,C 180,E1 -11641.505,E2 -11641.505} C_VEL
LIN {X 0,Y 390.086,Z 134.703,A -85,B 0,C 180,E1 -11645.207,E2 -11645.207} C_VEL
LIN {X 0,Y 390.07,Z 134.706,A -85,B 0,C 180,E1 -11649.218,E2 -11649.218} C_VEL
LIN {X 0,Y 390.043,Z 134.71,A -85,B 0,C 180,E1 -11652.374,E2 -11652.374} C_VEL
LIN {X 0,Y 390.044,Z 134.711,A -85,B 0,C 180,E1 -11655.354,E2 -11655.354} C_VEL
LIN {X 0,Y 390.031,Z 134.711,A -85,B 0,C 180,E1 -11658.187,E2 -11658.187} C_VEL
LIN {X 0,Y 390.088,Z 134.704,A -85,B 0,C 180,E1 -11660.908,E2 -11660.908} C_VEL
LIN {X 0,Y 390.086,Z 134.704,A -85,B 0,C 180,E1 -11664.793,E2 -11664.793} C_VEL
LIN {X 0,Y 390.024,Z 134.711,A -85,B 0,C 180,E1 -11668.496,E2 -11668.496} C_VEL
LIN {X 0,Y 390.118,Z 134.699,A -85,B 0,C 180,E1 -11672.07,E2 -11672.07} C_VEL
LIN {X 0,Y 390.081,Z 134.705,A -85,B 0,C 180,E1 -11675.519,E2 -11675.519} C_VEL
LIN {X 0,Y 390.057,Z 134.713,A -85,B 0,C 180,E1 -11678.878,E2 -11678.878} C_VEL
LIN {X 0,Y 390.129,Z 134.699,A -85,B 0,C 180,E1 -11682.167,E2 -11682.167} C_VEL
LIN {X 0,Y 390.145,Z 134.696,A -85,B 0,C 180,E1 -11685.393,E2 -11685.393} C_VEL
LIN {X 0,Y 390.15,Z 134.701,A -85,B 0,C 180,E1 -11688.571,E2 -11688.571} C_VEL
LIN {X 0,Y 390.309,Z 134.678,A -85,B 0,C 180,E1 -11692.032,E2 -11692.032} C_VEL
LIN {X 0,Y 390.226,Z 134.687,A -85,B 0,C 180,E1 -11694.834,E2 -11694.834} C_VEL
LIN {X 0,Y 390.419,Z 134.666,A -85,B 0,C 180,E1 -11697.937,E2 -11697.937} C_VEL
LIN {X 0,Y 390.55,Z 134.651,A -85,B 0,C 180,E1 -11700,E2 -11700} C_VEL
LIN {X 0,Y 390.311,Z 134.675,A -85,B 0,C 180,E1 -11703.097,E2 -11703.097} C_VEL
LIN {X 0,Y 390.312,Z 134.675,A -85,B 0,C 180,E1 -11706.627,E2 -11706.627} C_VEL
LIN {X 0,Y 390.212,Z 134.69,A -85,B 0,C 180,E1 -11709.329,E2 -11709.329} C_VEL
LIN {X 0,Y 390.18,Z 134.692,A -85,B 0,C 180,E1 -11712.483,E2 -11712.483} C_VEL
LIN {X 0,Y 390.142,Z 134.701,A -85,B 0,C 180,E1 -11715.677,E2 -11715.677} C_VEL
LIN {X 0,Y 390.107,Z 134.703,A -85,B 0,C 180,E1 -11718.922,E2 -11718.922} C_VEL
LIN {X 0,Y 390.041,Z 134.709,A -85,B 0,C 180,E1 -11722.234,E2 -11722.234} C_VEL
LIN {X 0,Y 390.121,Z 134.7,A -85,B 0,C 180,E1 -11725.743,E2 -11725.743} C_VEL
LIN {X 0,Y 390.061,Z 134.711,A -85,B 0,C 180,E1 -11729.109,E2 -11729.109} C_VEL
LIN {X 0,Y 390.044,Z 134.714,A -85,B 0,C 180,E1 -11732.721,E2 -11732.721} C_VEL
LIN {X 0,Y 390.058,Z 134.707,A -85,B 0,C 180,E1 -11735.825,E2 -11735.825} C_VEL
LIN {X 0,Y 390.069,Z 134.706,A -85,B 0,C 180,E1 -11739.218,E2 -11739.218} C_VEL
LIN {X 0,Y 390.044,Z 134.714,A -85,B 0,C 180,E1 -11742.374,E2 -11742.374} C_VEL
LIN {X 0,Y 390.046,Z 134.708,A -85,B 0,C 180,E1 -11745.354,E2 -11745.354} C_VEL
LIN {X 0,Y 390.033,Z 134.716,A -85,B 0,C 180,E1 -11748.187,E2 -11748.187} C_VEL
LIN {X 0,Y 390.094,Z 134.702,A -85,B 0,C 180,E1 -11750.908,E2 -11750.908} C_VEL
LIN {X 0,Y 390.087,Z 134.703,A -85,B 0,C 180,E1 -11754.793,E2 -11754.793} C_VEL
LIN {X 0,Y 390.034,Z 134.716,A -85,B 0,C 180,E1 -11757.875,E2 -11757.875} C_VEL
LIN {X 0,Y 390.06,Z 134.706,A -85,B 0,C 180,E1 -11760.89,E2 -11760.89} C_VEL
LIN {X 0,Y 390.121,Z 134.7,A -85,B 0,C 180,E1 -11764.257,E2 -11764.257} C_VEL
LIN {X 0,Y 390.123,Z 134.836,A -85,B 0,C 180,E1 -11768.292,E2 -11768.292} C_VEL
LIN {X 0,Y 391.077,Z 140.604,A -85,B 0,C 180,E1 -11770.035,E2 -11770.035} C_VEL
LIN {X 0,Y 390.895,Z 148.846,A -85,B 0,C 180,E1 -11772.346,E2 -11772.346} C_VEL
LIN {X 0,Y 390.553,Z 154.859,A -85,B 0,C 180,E1 -11773.938,E2 -11773.938} C_VEL
LIN {X 0,Y 390.951,Z 157.175,A -85,B 0,C 180,E1 -11774.052,E2 -11774.052} C_VEL
LIN {X 0,Y 393.934,Z 175.004,A -85,B 0,C 180,E1 -11774.508,E2 -11774.508} C_VEL
LIN {X 0,Y 393.373,Z 230.872,A -85,B 0,C 180,E1 -11775.548,E2 -11775.548} C_VEL
LIN {X 0,Y 393.093,Z 240.752,A -85,B 0,C 180,E1 -11775.868,E2 -11775.868} C_VEL
LIN {X 0,Y 392.716,Z 251.891,A -85,B 0,C 180,E1 -11776.415,E2 -11776.415} C_VEL
LIN {X 0,Y 392.146,Z 262.743,A -85,B 0,C 180,E1 -11777.186,E2 -11777.186} C_VEL
LIN {X 0,Y 391.592,Z 271.147,A -85,B 0,C 180,E1 -11777.957,E2 -11777.957} C_VEL
LIN {X 0,Y 391.076,Z 279.078,A -85,B 0,C 180,E1 -11778.861,E2 -11778.861} C_VEL
LIN {X 0,Y 390.648,Z 284.775,A -85,B 0,C 180,E1 -11779.635,E2 -11779.635} C_VEL
LIN {X 0,Y 390.089,Z 291.134,A -85,B 0,C 180,E1 -11780.668,E2 -11780.668} C_VEL
LIN {X 0,Y 389.63,Z 297.587,A -85,B 0,C 180,E1 -11781.964,E2 -11781.964} C_VEL
LIN {X 0,Y 389.409,Z 301.924,A -85,B 0,C 180,E1 -11783.041,E2 -11783.041} C_VEL
LIN {X 0,Y 389.126,Z 306.014,A -85,B 0,C 180,E1 -11784.299,E2 -11784.299} C_VEL
LIN {X 0,Y 388.931,Z 308.679,A -85,B 0,C 180,E1 -11785.336,E2 -11785.336} C_VEL
LIN {X 0,Y 388.745,Z 311.595,A -85,B 0,C 180,E1 -11786.891,E2 -11786.891} C_VEL
LIN {X 0,Y 388.699,Z 312.87,A -85,B 0,C 180,E1 -11787.927,E2 -11787.927} C_VEL
LIN {X 0,Y 388.675,Z 313.676,A -85,B 0,C 180,E1 -11788.964,E2 -11788.964} C_VEL
LIN {X 0,Y 388.672,Z 313.983,A -85,B 0,C 180,E1 -11790,E2 -11790} C_VEL
LIN {X 0,Y 388.675,Z 313.707,A -85,B 0,C 180,E1 -11791.036,E2 -11791.036} C_VEL
LIN {X 0,Y 388.698,Z 312.964,A -85,B 0,C 180,E1 -11792.072,E2 -11792.072} C_VEL
LIN {X 0,Y 388.741,Z 311.752,A -85,B 0,C 180,E1 -11793.109,E2 -11793.109} C_VEL
LIN {X 0,Y 388.923,Z 308.901,A -85,B 0,C 180,E1 -11794.664,E2 -11794.664} C_VEL
LIN {X 0,Y 389.108,Z 306.307,A -85,B 0,C 180,E1 -11795.701,E2 -11795.701} C_VEL
LIN {X 0,Y 389.378,Z 302.431,A -85,B 0,C 180,E1 -11796.921,E2 -11796.921} C_VEL
LIN {X 0,Y 389.607,Z 298.043,A -85,B 0,C 180,E1 -11798.036,E2 -11798.036} C_VEL
LIN {X 0,Y 389.951,Z 293.097,A -85,B 0,C 180,E1 -11799.073,E2 -11799.073} C_VEL
LIN {X 0,Y 390.443,Z 287.125,A -85,B 0,C 180,E1 -11800.108,E2 -11800.108} C_VEL
LIN {X 0,Y 390.572,Z 285.519,A -85,B 0,C 180,E1 -11800.352,E2 -11800.352} C_VEL
LIN {X 0,Y 390.267,Z 281.43,A -85,B 0,C 180,E1 -11800.964,E2 -11800.964} C_VEL
LIN {X 0,Y 388.036,Z 274.313,A -85,B 0,C 180,E1 -11801.92,E2 -11801.92} C_VEL
LIN {X 0,Y 385.741,Z 266.739,A -85,B 0,C 180,E1 -11802.791,E2 -11802.791} C_VEL
LIN {X 0,Y 385.356,Z 261.583,A -85,B 0,C 180,E1 -11803.259,E2 -11803.259} C_VEL
LIN {X 0,Y 385.967,Z 250.249,A -85,B 0,C 180,E1 -11804.028,E2 -11804.028} C_VEL
LIN {X 0,Y 386.348,Z 240.917,A -85,B 0,C 180,E1 -11804.485,E2 -11804.485} C_VEL
LIN {X 0,Y 386.589,Z 231.272,A -85,B 0,C 180,E1 -11804.806,E2 -11804.806} C_VEL
LIN {X 0,Y 387.048,Z 174.688,A -85,B 0,C 180,E1 -11805.886,E2 -11805.886} C_VEL
LIN {X 0,Y 383.633,Z 155.534,A -85,B 0,C 180,E1 -11806.411,E2 -11806.411} C_VEL
LIN {X 0,Y 383.637,Z 154.172,A -85,B 0,C 180,E1 -11806.633,E2 -11806.633} C_VEL
LIN {X 0,Y 384.106,Z 144.939,A -85,B 0,C 180,E1 -11809.229,E2 -11809.229} C_VEL
LIN {X 0,Y 384.022,Z 141.073,A -85,B 0,C 180,E1 -11810.348,E2 -11810.348} C_VEL
LIN {X 0,Y 383.086,Z 135.689,A -85,B 0,C 180,E1 -11812.02,E2 -11812.02} C_VEL
LIN {X 0,Y 383.08,Z 135.579,A -85,B 0,C 180,E1 -11816.123,E2 -11816.123} C_VEL
LIN {X 0,Y 383.041,Z 135.586,A -85,B 0,C 180,E1 -11818.492,E2 -11818.492} C_VEL
LIN {X 0,Y 383.01,Z 135.591,A -85,B 0,C 180,E1 -11822.149,E2 -11822.149} C_VEL
LIN {X 0,Y 383.018,Z 135.585,A -85,B 0,C 180,E1 -11824.667,E2 -11824.667} C_VEL
LIN {X 0,Y 383.001,Z 135.592,A -85,B 0,C 180,E1 -11827.904,E2 -11827.904} C_VEL
LIN {X 0,Y 382.984,Z 135.59,A -85,B 0,C 180,E1 -11831.347,E2 -11831.347} C_VEL
LIN {X 0,Y 382.995,Z 135.588,A -85,B 0,C 180,E1 -11834.303,E2 -11834.303} C_VEL
LIN {X 0,Y 383.009,Z 135.587,A -85,B 0,C 180,E1 -11837.24,E2 -11837.24} C_VEL
LIN {X 0,Y 383.012,Z 135.584,A -85,B 0,C 180,E1 -11840.413,E2 -11840.413} C_VEL
LIN {X 0,Y 383.024,Z 135.583,A -85,B 0,C 180,E1 -11844.044,E2 -11844.044} C_VEL
LIN {X 0,Y 382.985,Z 135.59,A -85,B 0,C 180,E1 -11847.578,E2 -11847.578} C_VEL
LIN {X 0,Y 382.991,Z 135.587,A -85,B 0,C 180,E1 -11850.3,E2 -11850.3} C_VEL
LIN {X 0,Y 383.079,Z 135.576,A -85,B 0,C 180,E1 -11854.021,E2 -11854.021} C_VEL
LIN {X 0,Y 383.007,Z 135.587,A -85,B 0,C 180,E1 -11857.335,E2 -11857.335} C_VEL
LIN {X 0,Y 383.059,Z 135.585,A -85,B 0,C 180,E1 -11860.716,E2 -11860.716} C_VEL
LIN {X 0,Y 383.08,Z 135.577,A -85,B 0,C 180,E1 -11864.026,E2 -11864.026} C_VEL
LIN {X 0,Y 383.14,Z 135.569,A -85,B 0,C 180,E1 -11867.284,E2 -11867.284} C_VEL
LIN {X 0,Y 383.155,Z 135.571,A -85,B 0,C 180,E1 -11870.498,E2 -11870.498} C_VEL
LIN {X 0,Y 383.272,Z 135.555,A -85,B 0,C 180,E1 -11872.625,E2 -11872.625} C_VEL
LIN {X 0,Y 383.197,Z 135.563,A -85,B 0,C 180,E1 -11874.738,E2 -11874.738} C_VEL
LIN {X 0,Y 383.386,Z 135.543,A -85,B 0,C 180,E1 -11877.899,E2 -11877.899} C_VEL
LIN {X 0,Y 383.518,Z 135.528,A -85,B 0,C 180,E1 -11880,E2 -11880} C_VEL
LIN {X 0,Y 383.246,Z 135.556,A -85,B 0,C 180,E1 -11883.154,E2 -11883.154} C_VEL
LIN {X 0,Y 383.292,Z 135.551,A -85,B 0,C 180,E1 -11886.316,E2 -11886.316} C_VEL
LIN {X 0,Y 383.258,Z 135.554,A -85,B 0,C 180,E1 -11888.436,E2 -11888.436} C_VEL
LIN {X 0,Y 383.096,Z 135.579,A -85,B 0,C 180,E1 -11891.642,E2 -11891.642} C_VEL
LIN {X 0,Y 383.108,Z 135.574,A -85,B 0,C 180,E1 -11894.882,E2 -11894.882} C_VEL
LIN {X 0,Y 383.061,Z 135.578,A -85,B 0,C 180,E1 -11898.174,E2 -11898.174} C_VEL
LIN {X 0,Y 382.991,Z 135.59,A -85,B 0,C 180,E1 -11901.531,E2 -11901.531} C_VEL
LIN {X 0,Y 383.05,Z 135.586,A -85,B 0,C 180,E1 -11904.96,E2 -11904.96} C_VEL
LIN {X 0,Y 383.038,Z 135.584,A -85,B 0,C 180,E1 -11908.493,E2 -11908.493} C_VEL
LIN {X 0,Y 383.007,Z 135.586,A -85,B 0,C 180,E1 -11912.15,E2 -11912.15} C_VEL
LIN {X 0,Y 383.016,Z 135.59,A -85,B 0,C 180,E1 -11914.668,E2 -11914.668} C_VEL
LIN {X 0,Y 382.996,Z 135.587,A -85,B 0,C 180,E1 -11917.904,E2 -11917.904} C_VEL
LIN {X 0,Y 382.981,Z 135.588,A -85,B 0,C 180,E1 -11921.348,E2 -11921.348} C_VEL
LIN {X 0,Y 382.994,Z 135.593,A -85,B 0,C 180,E1 -11924.304,E2 -11924.304} C_VEL
LIN {X 0,Y 383.008,Z 135.585,A -85,B 0,C 180,E1 -11927.24,E2 -11927.24} C_VEL
LIN {X 0,Y 383.013,Z 135.587,A -85,B 0,C 180,E1 -11930.414,E2 -11930.414} C_VEL
LIN {X 0,Y 383.024,Z 135.588,A -85,B 0,C 180,E1 -11934.045,E2 -11934.045} C_VEL
LIN {X 0,Y 382.986,Z 135.592,A -85,B 0,C 180,E1 -11937.578,E2 -11937.578} C_VEL
LIN {X 0,Y 382.991,Z 135.588,A -85,B 0,C 180,E1 -11940.3,E2 -11940.3} C_VEL
LIN {X 0,Y 383.056,Z 135.579,A -85,B 0,C 180,E1 -11942.698,E2 -11942.698} C_VEL
LIN {X 0,Y 383.108,Z 135.637,A -85,B 0,C 180,E1 -11944.899,E2 -11944.899} C_VEL
LIN {X 0,Y 384.634,Z 144.418,A -85,B 0,C 180,E1 -11947.437,E2 -11947.437} C_VEL
LIN {X 0,Y 384.773,Z 148.621,A -85,B 0,C 180,E1 -11948.574,E2 -11948.574} C_VEL
LIN {X 0,Y 383.701,Z 162.711,A -85,B 0,C 180,E1 -11952.26,E2 -11952.26} C_VEL
LIN {X 0,Y 383.446,Z 167.905,A -85,B 0,C 180,E1 -11953.564,E2 -11953.564} C_VEL
LIN {X 0,Y 384.012,Z 171.982,A -85,B 0,C 180,E1 -11953.723,E2 -11953.723} C_VEL
LIN {X 0,Y 386.995,Z 193.588,A -85,B 0,C 180,E1 -11954.26,E2 -11954.26} C_VEL
LIN {X 0,Y 386.474,Z 244.39,A -85,B 0,C 180,E1 -11955.224,E2 -11955.224} C_VEL
LIN {X 0,Y 386.137,Z 253.336,A -85,B 0,C 180,E1 -11955.507,E2 -11955.507} C_VEL
LIN {X 0,Y 385.675,Z 262.983,A -85,B 0,C 180,E1 -11955.961,E2 -11955.961} C_VEL
LIN {X 0,Y 385.174,Z 272.135,A -85,B 0,C 180,E1 -11956.548,E2 -11956.548} C_VEL
LIN {X 0,Y 384.45,Z 282.928,A -85,B 0,C 180,E1 -11957.463,E2 -11957.463} C_VEL
LIN {X 0,Y 383.79,Z 292.234,A -85,B 0,C 180,E1 -11958.513,E2 -11958.513} C_VEL
LIN {X 0,Y 383.23,Z 298.902,A -85,B 0,C 180,E1 -11959.433,E2 -11959.433} C_VEL
LIN {X 0,Y 382.765,Z 305.233,A -85,B 0,C 180,E1 -11960.489,E2 -11960.489} C_VEL
LIN {X 0,Y 382.373,Z 310.493,A -85,B 0,C 180,E1 -11961.545,E2 -11961.545} C_VEL
LIN {X 0,Y 382.067,Z 314.88,A -85,B 0,C 180,E1 -11962.602,E2 -11962.602} C_VEL
LIN {X 0,Y 381.772,Z 319.754,A -85,B 0,C 180,E1 -11964.085,E2 -11964.085} C_VEL
LIN {X 0,Y 381.714,Z 322.698,A -85,B 0,C 180,E1 -11965.248,E2 -11965.248} C_VEL
LIN {X 0,Y 381.538,Z 325.597,A -85,B 0,C 180,E1 -11966.832,E2 -11966.832} C_VEL
LIN {X 0,Y 381.533,Z 326.848,A -85,B 0,C 180,E1 -11967.889,E2 -11967.889} C_VEL
LIN {X 0,Y 381.554,Z 327.626,A -85,B 0,C 180,E1 -11968.945,E2 -11968.945} C_VEL
LIN {X 0,Y 381.586,Z 327.921,A -85,B 0,C 180,E1 -11970,E2 -11970} C_VEL
LIN {X 0,Y 381.554,Z 327.622,A -85,B 0,C 180,E1 -11971.056,E2 -11971.056} C_VEL
LIN {X 0,Y 381.533,Z 326.837,A -85,B 0,C 180,E1 -11972.112,E2 -11972.112} C_VEL
LIN {X 0,Y 381.539,Z 325.579,A -85,B 0,C 180,E1 -11973.168,E2 -11973.168} C_VEL
LIN {X 0,Y 381.714,Z 322.673,A -85,B 0,C 180,E1 -11974.753,E2 -11974.753} C_VEL
LIN {X 0,Y 381.771,Z 319.724,A -85,B 0,C 180,E1 -11975.915,E2 -11975.915} C_VEL
LIN {X 0,Y 382.057,Z 314.836,A -85,B 0,C 180,E1 -11977.399,E2 -11977.399} C_VEL
LIN {X 0,Y 382.527,Z 308.004,A -85,B 0,C 180,E1 -11978.985,E2 -11978.985} C_VEL
LIN {X 0,Y 383.112,Z 300.537,A -85,B 0,C 180,E1 -11980.304,E2 -11980.304} C_VEL
LIN {X 0,Y 383.723,Z 293.174,A -85,B 0,C 180,E1 -11981.355,E2 -11981.355} C_VEL
LIN {X 0,Y 384.267,Z 285.287,A -85,B 0,C 180,E1 -11982.276,E2 -11982.276} C_VEL
LIN {X 0,Y 384.845,Z 276.952,A -85,B 0,C 180,E1 -11983.061,E2 -11983.061} C_VEL
LIN {X 0,Y 385.528,Z 266.305,A -85,B 0,C 180,E1 -11983.843,E2 -11983.843} C_VEL
LIN {X 0,Y 386.053,Z 254.706,A -85,B 0,C 180,E1 -11984.429,E2 -11984.429} C_VEL
LIN {X 0,Y 386.409,Z 244.981,A -85,B 0,C 180,E1 -11984.752,E2 -11984.752} C_VEL
LIN {X 0,Y 386.911,Z 191.571,A -85,B 0,C 180,E1 -11985.77,E2 -11985.77} C_VEL
LIN {X 0,Y 383.454,Z 168.193,A -85,B 0,C 180,E1 -11986.392,E2 -11986.392} C_VEL
LIN {X 0,Y 383.628,Z 163.992,A -85,B 0,C 180,E1 -11987.394,E2 -11987.394} C_VEL
LIN {X 0,Y 384.601,Z 150.899,A -85,B 0,C 180,E1 -11990.813,E2 -11990.813} C_VEL
LIN {X 0,Y 384.778,Z 145.418,A -85,B 0,C 180,E1 -11992.272,E2 -11992.272} C_VEL
LIN {X 0,Y 383.11,Z 135.619,A -85,B 0,C 180,E1 -11995.101,E2 -11995.101} C_VEL
LIN {X 0,Y 383.041,Z 135.586,A -85,B 0,C 180,E1 -11998.493,E2 -11998.493} C_VEL
LIN {X 0,Y 383.01,Z 135.59,A -85,B 0,C 180,E1 -12002.15,E2 -12002.15} C_VEL
LIN {X 0,Y 383.019,Z 135.585,A -85,B 0,C 180,E1 -12004.668,E2 -12004.668} C_VEL
LIN {X 0,Y 383,Z 135.591,A -85,B 0,C 180,E1 -12007.904,E2 -12007.904} C_VEL
LIN {X 0,Y 382.984,Z 135.589,A -85,B 0,C 180,E1 -12011.348,E2 -12011.348} C_VEL
LIN {X 0,Y 382.996,Z 135.588,A -85,B 0,C 180,E1 -12014.303,E2 -12014.303} C_VEL
LIN {X 0,Y 383.011,Z 135.587,A -85,B 0,C 180,E1 -12017.24,E2 -12017.24} C_VEL
LIN {X 0,Y 383.014,Z 135.584,A -85,B 0,C 180,E1 -12020.414,E2 -12020.414} C_VEL
LIN {X 0,Y 383.026,Z 135.584,A -85,B 0,C 180,E1 -12024.045,E2 -12024.045} C_VEL
LIN {X 0,Y 382.987,Z 135.591,A -85,B 0,C 180,E1 -12027.578,E2 -12027.578} C_VEL
LIN {X 0,Y 382.993,Z 135.587,A -85,B 0,C 180,E1 -12030.3,E2 -12030.3} C_VEL
LIN {X 0,Y 383.058,Z 135.581,A -85,B 0,C 180,E1 -12032.698,E2 -12032.698} C_VEL
LIN {X 0,Y 383.053,Z 135.586,A -85,B 0,C 180,E1 -12035.04,E2 -12035.04} C_VEL
LIN {X 0,Y 382.994,Z 135.589,A -85,B 0,C 180,E1 -12038.469,E2 -12038.469} C_VEL
LIN {X 0,Y 383.064,Z 135.578,A -85,B 0,C 180,E1 -12041.827,E2 -12041.827} C_VEL
LIN {X 0,Y 383.112,Z 135.574,A -85,B 0,C 180,E1 -12045.118,E2 -12045.118} C_VEL
LIN {X 0,Y 383.099,Z 135.578,A -85,B 0,C 180,E1 -12048.358,E2 -12048.358} C_VEL
LIN {X 0,Y 383.265,Z 135.555,A -85,B 0,C 180,E1 -12051.976,E2 -12051.976} C_VEL
LIN {X 0,Y 383.198,Z 135.563,A -85,B 0,C 180,E1 -12054.739,E2 -12054.739} C_VEL
LIN {X 0,Y 383.387,Z 135.541,A -85,B 0,C 180,E1 -12057.899,E2 -12057.899} C_VEL
LIN {X 0,Y 383.519,Z 135.527,A -85,B 0,C 180,E1 -12060,E2 -12060} C_VEL
LIN {X 0,Y 383.247,Z 135.555,A -85,B 0,C 180,E1 -12063.154,E2 -12063.154} C_VEL
LIN {X 0,Y 383.272,Z 135.552,A -85,B 0,C 180,E1 -12066.621,E2 -12066.621} C_VEL
LIN {X 0,Y 383.263,Z 135.554,A -85,B 0,C 180,E1 -12068.436,E2 -12068.436} C_VEL
LIN {X 0,Y 383.11,Z 135.579,A -85,B 0,C 180,E1 -12071.642,E2 -12071.642} C_VEL
LIN {X 0,Y 383.114,Z 135.573,A -85,B 0,C 180,E1 -12074.882,E2 -12074.882} C_VEL
LIN {X 0,Y 383.065,Z 135.578,A -85,B 0,C 180,E1 -12078.174,E2 -12078.174} C_VEL
LIN {X 0,Y 382.995,Z 135.59,A -85,B 0,C 180,E1 -12081.531,E2 -12081.531} C_VEL
LIN {X 0,Y 383.054,Z 135.584,A -85,B 0,C 180,E1 -12084.96,E2 -12084.96} C_VEL
LIN {X 0,Y 383.042,Z 135.582,A -85,B 0,C 180,E1 -12088.493,E2 -12088.493} C_VEL
LIN {X 0,Y 383.011,Z 135.585,A -85,B 0,C 180,E1 -12092.15,E2 -12092.15} C_VEL
LIN {X 0,Y 383.02,Z 135.589,A -85,B 0,C 180,E1 -12094.668,E2 -12094.668} C_VEL
LIN {X 0,Y 383,Z 135.586,A -85,B 0,C 180,E1 -12097.903,E2 -12097.903} C_VEL
LIN {X 0,Y 382.985,Z 135.588,A -85,B 0,C 180,E1 -12101.347,E2 -12101.347} C_VEL
LIN {X 0,Y 382.997,Z 135.592,A -85,B 0,C 180,E1 -12104.303,E2 -12104.303} C_VEL
LIN {X 0,Y 383.012,Z 135.584,A -85,B 0,C 180,E1 -12107.24,E2 -12107.24} C_VEL
LIN {X 0,Y 383.018,Z 135.587,A -85,B 0,C 180,E1 -12110.413,E2 -12110.413} C_VEL
LIN {X 0,Y 383.028,Z 135.589,A -85,B 0,C 180,E1 -12114.045,E2 -12114.045} C_VEL
LIN {X 0,Y 382.989,Z 135.59,A -85,B 0,C 180,E1 -12117.578,E2 -12117.578} C_VEL
LIN {X 0,Y 382.994,Z 135.588,A -85,B 0,C 180,E1 -12120.3,E2 -12120.3} C_VEL
LIN {X 0,Y 383.058,Z 135.579,A -85,B 0,C 180,E1 -12122.698,E2 -12122.698} C_VEL
LIN {X 0,Y 383.053,Z 135.58,A -85,B 0,C 180,E1 -12125.04,E2 -12125.04} C_VEL
LIN {X 0,Y 383.096,Z 135.755,A -85,B 0,C 180,E1 -12128.121,E2 -12128.121} C_VEL
LIN {X 0,Y 384.14,Z 142.642,A -85,B 0,C 180,E1 -12130.216,E2 -12130.216} C_VEL
LIN {X 0,Y 383.746,Z 152.341,A -85,B 0,C 180,E1 -12132.961,E2 -12132.961} C_VEL
LIN {X 0,Y 383.611,Z 154.986,A -85,B 0,C 180,E1 -12133.639,E2 -12133.639} C_VEL
LIN {X 0,Y 384.018,Z 157.527,A -85,B 0,C 180,E1 -12133.76,E2 -12133.76} C_VEL
LIN {X 0,Y 387.109,Z 176.027,A -85,B 0,C 180,E1 -12134.244,E2 -12134.244} C_VEL
LIN {X 0,Y 386.516,Z 231.019,A -85,B 0,C 180,E1 -12135.286,E2 -12135.286} C_VEL
LIN {X 0,Y 386.223,Z 240.892,A -85,B 0,C 180,E1 -12135.611,E2 -12135.611} C_VEL
LIN {X 0,Y 385.837,Z 252.027,A -85,B 0,C 180,E1 -12136.168,E2 -12136.168} C_VEL
LIN {X 0,Y 385.243,Z 262.877,A -85,B 0,C 180,E1 -12136.952,E2 -12136.952} C_VEL
LIN {X 0,Y 384.667,Z 271.28,A -85,B 0,C 180,E1 -12137.737,E2 -12137.737} C_VEL
LIN {X 0,Y 384.118,Z 279.21,A -85,B 0,C 180,E1 -12138.656,E2 -12138.656} C_VEL
LIN {X 0,Y 383.678,Z 284.906,A -85,B 0,C 180,E1 -12139.445,E2 -12139.445} C_VEL
LIN {X 0,Y 383.097,Z 291.265,A -85,B 0,C 180,E1 -12140.496,E2 -12140.496} C_VEL
LIN {X 0,Y 382.702,Z 296.548,A -85,B 0,C 180,E1 -12141.552,E2 -12141.552} C_VEL
LIN {X 0,Y 382.433,Z 300.958,A -85,B 0,C 180,E1 -12142.609,E2 -12142.609} C_VEL
LIN {X 0,Y 382.168,Z 304.632,A -85,B 0,C 180,E1 -12143.665,E2 -12143.665} C_VEL
LIN {X 0,Y 381.99,Z 307.631,A -85,B 0,C 180,E1 -12144.722,E2 -12144.722} C_VEL
LIN {X 0,Y 381.777,Z 309.955,A -85,B 0,C 180,E1 -12145.777,E2 -12145.777} C_VEL
LIN {X 0,Y 381.654,Z 311.724,A -85,B 0,C 180,E1 -12146.833,E2 -12146.833} C_VEL
LIN {X 0,Y 381.601,Z 312.999,A -85,B 0,C 180,E1 -12147.889,E2 -12147.889} C_VEL
LIN {X 0,Y 381.576,Z 313.805,A -85,B 0,C 180,E1 -12148.944,E2 -12148.944} C_VEL
LIN {X 0,Y 381.587,Z 314.111,A -85,B 0,C 180,E1 -12150,E2 -12150} C_VEL
LIN {X 0,Y 381.576,Z 313.835,A -85,B 0,C 180,E1 -12151.055,E2 -12151.055} C_VEL
LIN {X 0,Y 381.601,Z 313.092,A -85,B 0,C 180,E1 -12152.111,E2 -12152.111} C_VEL
LIN {X 0,Y 381.65,Z 311.88,A -85,B 0,C 180,E1 -12153.167,E2 -12153.167} C_VEL
LIN {X 0,Y 381.864,Z 309.028,A -85,B 0,C 180,E1 -12154.75,E2 -12154.75} C_VEL
LIN {X 0,Y 382.047,Z 306.434,A -85,B 0,C 180,E1 -12155.807,E2 -12155.807} C_VEL
LIN {X 0,Y 382.42,Z 301.326,A -85,B 0,C 180,E1 -12157.391,E2 -12157.391} C_VEL
LIN {X 0,Y 382.757,Z 295.831,A -85,B 0,C 180,E1 -12158.713,E2 -12158.713} C_VEL
LIN {X 0,Y 383.339,Z 288.928,A -85,B 0,C 180,E1 -12160.03,E2 -12160.03} C_VEL
LIN {X 0,Y 383.97,Z 281,A -85,B 0,C 180,E1 -12161.214,E2 -12161.214} C_VEL
LIN {X 0,Y 384.534,Z 273.439,A -85,B 0,C 180,E1 -12162.133,E2 -12162.133} C_VEL
LIN {X 0,Y 384.972,Z 267.013,A -85,B 0,C 180,E1 -12162.788,E2 -12162.788} C_VEL
LIN {X 0,Y 385.356,Z 261.583,A -85,B 0,C 180,E1 -12163.259,E2 -12163.259} C_VEL
LIN {X 0,Y 384.907,Z 256.421,A -85,B 0,C 180,E1 -12163.694,E2 -12163.694} C_VEL
LIN {X 0,Y 382.391,Z 247.796,A -85,B 0,C 180,E1 -12164.345,E2 -12164.345} C_VEL
LIN {X 0,Y 380.335,Z 240.649,A -85,B 0,C 180,E1 -12164.761,E2 -12164.761} C_VEL
LIN {X 0,Y 379.678,Z 234.993,A -85,B 0,C 180,E1 -12164.985,E2 -12164.985} C_VEL
LIN {X 0,Y 379.69,Z 233.061,A -85,B 0,C 180,E1 -12165.037,E2 -12165.037} C_VEL
LIN {X 0,Y 379.901,Z 211.592,A -85,B 0,C 180,E1 -12165.484,E2 -12165.484} C_VEL
LIN {X 0,Y 380.224,Z 175.493,A -85,B 0,C 180,E1 -12166.165,E2 -12166.165} C_VEL
LIN {X 0,Y 376.694,Z 155.45,A -85,B 0,C 180,E1 -12166.739,E2 -12166.739} C_VEL
LIN {X 0,Y 376.664,Z 154.294,A -85,B 0,C 180,E1 -12166.95,E2 -12166.95} C_VEL
LIN {X 0,Y 377.128,Z 145.05,A -85,B 0,C 180,E1 -12169.599,E2 -12169.599} C_VEL
LIN {X 0,Y 376.675,Z 140.015,A -85,B 0,C 180,E1 -12171.108,E2 -12171.108} C_VEL
LIN {X 0,Y 376.026,Z 136.561,A -85,B 0,C 180,E1 -12172.239,E2 -12172.239} C_VEL
LIN {X 0,Y 376.042,Z 136.457,A -85,B 0,C 180,E1 -12176.221,E2 -12176.221} C_VEL
LIN {X 0,Y 375.97,Z 136.462,A -85,B 0,C 180,E1 -12179.079,E2 -12179.079} C_VEL
LIN {X 0,Y 375.951,Z 136.465,A -85,B 0,C 180,E1 -12182.828,E2 -12182.828} C_VEL
LIN {X 0,Y 375.958,Z 136.464,A -85,B 0,C 180,E1 -12185.415,E2 -12185.415} C_VEL
LIN {X 0,Y 375.976,Z 136.464,A -85,B 0,C 180,E1 -12188.27,E2 -12188.27} C_VEL
LIN {X 0,Y 375.934,Z 136.47,A -85,B 0,C 180,E1 -12191.6,E2 -12191.6} C_VEL
LIN {X 0,Y 375.926,Z 136.469,A -85,B 0,C 180,E1 -12195.268,E2 -12195.268} C_VEL
LIN {X 0,Y 375.933,Z 136.466,A -85,B 0,C 180,E1 -12198.399,E2 -12198.399} C_VEL
LIN {X 0,Y 375.971,Z 136.465,A -85,B 0,C 180,E1 -12201.729,E2 -12201.729} C_VEL
LIN {X 0,Y 375.979,Z 136.467,A -85,B 0,C 180,E1 -12205.332,E2 -12205.332} C_VEL
LIN {X 0,Y 375.956,Z 136.464,A -85,B 0,C 180,E1 -12208.438,E2 -12208.438} C_VEL
LIN {X 0,Y 375.982,Z 136.46,A -85,B 0,C 180,E1 -12212.14,E2 -12212.14} C_VEL
LIN {X 0,Y 376.005,Z 136.46,A -85,B 0,C 180,E1 -12214.539,E2 -12214.539} C_VEL
LIN {X 0,Y 375.962,Z 136.463,A -85,B 0,C 180,E1 -12218.046,E2 -12218.046} C_VEL
LIN {X 0,Y 376.008,Z 136.457,A -85,B 0,C 180,E1 -12221.473,E2 -12221.473} C_VEL
LIN {X 0,Y 376.058,Z 136.454,A -85,B 0,C 180,E1 -12224.832,E2 -12224.832} C_VEL
LIN {X 0,Y 376.058,Z 136.454,A -85,B 0,C 180,E1 -12228.137,E2 -12228.137} C_VEL
LIN {X 0,Y 376.256,Z 136.428,A -85,B 0,C 180,E1 -12231.877,E2 -12231.877} C_VEL
LIN {X 0,Y 376.17,Z 136.439,A -85,B 0,C 180,E1 -12234.64,E2 -12234.64} C_VEL
LIN {X 0,Y 376.352,Z 136.418,A -85,B 0,C 180,E1 -12237.86,E2 -12237.86} C_VEL
LIN {X 0,Y 376.487,Z 136.403,A -85,B 0,C 180,E1 -12240,E2 -12240} C_VEL
LIN {X 0,Y 376.184,Z 136.436,A -85,B 0,C 180,E1 -12243.213,E2 -12243.213} C_VEL
LIN {X 0,Y 376.251,Z 136.427,A -85,B 0,C 180,E1 -12246.435,E2 -12246.435} C_VEL
LIN {X 0,Y 376.204,Z 136.433,A -85,B 0,C 180,E1 -12248.595,E2 -12248.595} C_VEL
LIN {X 0,Y 376.049,Z 136.455,A -85,B 0,C 180,E1 -12251.863,E2 -12251.863} C_VEL
LIN {X 0,Y 376.056,Z 136.455,A -85,B 0,C 180,E1 -12255.167,E2 -12255.167} C_VEL
LIN {X 0,Y 376.007,Z 136.457,A -85,B 0,C 180,E1 -12258.527,E2 -12258.527} C_VEL
LIN {X 0,Y 375.961,Z 136.463,A -85,B 0,C 180,E1 -12261.954,E2 -12261.954} C_VEL
LIN {X 0,Y 376.004,Z 136.459,A -85,B 0,C 180,E1 -12265.461,E2 -12265.461} C_VEL
LIN {X 0,Y 375.968,Z 136.466,A -85,B 0,C 180,E1 -12269.079,E2 -12269.079} C_VEL
LIN {X 0,Y 375.947,Z 136.47,A -85,B 0,C 180,E1 -12272.829,E2 -12272.829} C_VEL
LIN {X 0,Y 375.955,Z 136.464,A -85,B 0,C 180,E1 -12275.416,E2 -12275.416} C_VEL
LIN {X 0,Y 375.97,Z 136.465,A -85,B 0,C 180,E1 -12278.27,E2 -12278.27} C_VEL
LIN {X 0,Y 375.932,Z 136.467,A -85,B 0,C 180,E1 -12281.601,E2 -12281.601} C_VEL
LIN {X 0,Y 375.925,Z 136.467,A -85,B 0,C 180,E1 -12285.269,E2 -12285.269} C_VEL
LIN {X 0,Y 375.932,Z 136.47,A -85,B 0,C 180,E1 -12288.399,E2 -12288.399} C_VEL
LIN {X 0,Y 375.972,Z 136.465,A -85,B 0,C 180,E1 -12291.73,E2 -12291.73} C_VEL
LIN {X 0,Y 375.979,Z 136.462,A -85,B 0,C 180,E1 -12295.333,E2 -12295.333} C_VEL
LIN {X 0,Y 375.956,Z 136.464,A -85,B 0,C 180,E1 -12298.438,E2 -12298.438} C_VEL
LIN {X 0,Y 375.995,Z 136.46,A -85,B 0,C 180,E1 -12302.142,E2 -12302.142} C_VEL
LIN {X 0,Y 376.059,Z 136.533,A -85,B 0,C 180,E1 -12304.691,E2 -12304.691} C_VEL
LIN {X 0,Y 377.768,Z 146.394,A -85,B 0,C 180,E1 -12307.581,E2 -12307.581} C_VEL
LIN {X 0,Y 377.666,Z 151.128,A -85,B 0,C 180,E1 -12308.87,E2 -12308.87} C_VEL
LIN {X 0,Y 376.531,Z 166.289,A -85,B 0,C 180,E1 -12312.904,E2 -12312.904} C_VEL
LIN {X 0,Y 376.467,Z 168.14,A -85,B 0,C 180,E1 -12313.286,E2 -12313.286} C_VEL
LIN {X 0,Y 380.129,Z 192.997,A -85,B 0,C 180,E1 -12313.958,E2 -12313.958} C_VEL
LIN {X 0,Y 379.62,Z 244.324,A -85,B 0,C 180,E1 -12314.952,E2 -12314.952} C_VEL
LIN {X 0,Y 379.265,Z 254.049,A -85,B 0,C 180,E1 -12315.273,E2 -12315.273} C_VEL
LIN {X 0,Y 378.738,Z 264.072,A -85,B 0,C 180,E1 -12315.767,E2 -12315.767} C_VEL
LIN {X 0,Y 378.049,Z 275.458,A -85,B 0,C 180,E1 -12316.563,E2 -12316.563} C_VEL
LIN {X 0,Y 377.39,Z 284.035,A -85,B 0,C 180,E1 -12317.361,E2 -12317.361} C_VEL
LIN {X 0,Y 376.823,Z 292.108,A -85,B 0,C 180,E1 -12318.298,E2 -12318.298} C_VEL
LIN {X 0,Y 376.236,Z 298.775,A -85,B 0,C 180,E1 -12319.234,E2 -12319.234} C_VEL
LIN {X 0,Y 375.764,Z 305.106,A -85,B 0,C 180,E1 -12320.31,E2 -12320.31} C_VEL
LIN {X 0,Y 375.346,Z 310.366,A -85,B 0,C 180,E1 -12321.385,E2 -12321.385} C_VEL
LIN {X 0,Y 375.012,Z 314.753,A -85,B 0,C 180,E1 -12322.462,E2 -12322.462} C_VEL
LIN {X 0,Y 374.668,Z 320.103,A -85,B 0,C 180,E1 -12324.142,E2 -12324.142} C_VEL
LIN {X 0,Y 374.603,Z 323.725,A -85,B 0,C 180,E1 -12325.696,E2 -12325.696} C_VEL
LIN {X 0,Y 374.456,Z 325.469,A -85,B 0,C 180,E1 -12326.772,E2 -12326.772} C_VEL
LIN {X 0,Y 374.432,Z 326.72,A -85,B 0,C 180,E1 -12327.849,E2 -12327.849} C_VEL
LIN {X 0,Y 374.454,Z 327.498,A -85,B 0,C 180,E1 -12328.925,E2 -12328.925} C_VEL
LIN {X 0,Y 374.487,Z 327.792,A -85,B 0,C 180,E1 -12330,E2 -12330} C_VEL
LIN {X 0,Y 374.454,Z 327.494,A -85,B 0,C 180,E1 -12331.076,E2 -12331.076} C_VEL
LIN {X 0,Y 374.432,Z 326.708,A -85,B 0,C 180,E1 -12332.152,E2 -12332.152} C_VEL
LIN {X 0,Y 374.456,Z 325.451,A -85,B 0,C 180,E1 -12333.228,E2 -12333.228} C_VEL
LIN {X 0,Y 374.631,Z 322.543,A -85,B 0,C 180,E1 -12334.843,E2 -12334.843} C_VEL
LIN {X 0,Y 374.743,Z 318.837,A -85,B 0,C 180,E1 -12336.295,E2 -12336.295} C_VEL
LIN {X 0,Y 375.04,Z 313.744,A -85,B 0,C 180,E1 -12337.809,E2 -12337.809} C_VEL
LIN {X 0,Y 375.513,Z 307.874,A -85,B 0,C 180,E1 -12339.154,E2 -12339.154} C_VEL
LIN {X 0,Y 376.117,Z 300.406,A -85,B 0,C 180,E1 -12340.497,E2 -12340.497} C_VEL
LIN {X 0,Y 376.762,Z 293.043,A -85,B 0,C 180,E1 -12341.568,E2 -12341.568} C_VEL
LIN {X 0,Y 377.322,Z 285.155,A -85,B 0,C 180,E1 -12342.505,E2 -12342.505} C_VEL
LIN {X 0,Y 377.941,Z 276.82,A -85,B 0,C 180,E1 -12343.304,E2 -12343.304} C_VEL
LIN {X 0,Y 378.641,Z 266.171,A -85,B 0,C 180,E1 -12344.1,E2 -12344.1} C_VEL
LIN {X 0,Y 379.19,Z 254.568,A -85,B 0,C 180,E1 -12344.696,E2 -12344.696} C_VEL
LIN {X 0,Y 379.567,Z 244.838,A -85,B 0,C 180,E1 -12345.024,E2 -12345.024} C_VEL
LIN {X 0,Y 379.996,Z 191.778,A -85,B 0,C 180,E1 -12346.058,E2 -12346.058} C_VEL
LIN {X 0,Y 376.46,Z 168.058,A -85,B 0,C 180,E1 -12346.705,E2 -12346.705} C_VEL
LIN {X 0,Y 376.656,Z 163.762,A -85,B 0,C 180,E1 -12347.754,E2 -12347.754} C_VEL
LIN {X 0,Y 377.675,Z 151.111,A -85,B 0,C 180,E1 -12351.12,E2 -12351.12} C_VEL
LIN {X 0,Y 377.761,Z 146.338,A -85,B 0,C 180,E1 -12352.42,E2 -12352.42} C_VEL
LIN {X 0,Y 376.061,Z 136.515,A -85,B 0,C 180,E1 -12355.309,E2 -12355.309} C_VEL
LIN {X 0,Y 375.971,Z 136.462,A -85,B 0,C 180,E1 -12359.079,E2 -12359.079} C_VEL
LIN {X 0,Y 375.95,Z 136.465,A -85,B 0,C 180,E1 -12362.829,E2 -12362.829} C_VEL
LIN {X 0,Y 375.958,Z 136.464,A -85,B 0,C 180,E1 -12365.416,E2 -12365.416} C_VEL
LIN {X 0,Y 375.974,Z 136.465,A -85,B 0,C 180,E1 -12368.271,E2 -12368.271} C_VEL
LIN {X 0,Y 375.935,Z 136.469,A -85,B 0,C 180,E1 -12371.601,E2 -12371.601} C_VEL
LIN {X 0,Y 375.927,Z 136.469,A -85,B 0,C 180,E1 -12375.269,E2 -12375.269} C_VEL
